   1:  PR[91,1] = PR[90,1] + 61.164;
   1:  PR[91,2] = PR[90,2] + 21.945;
   1:  PR[91,3] = PR[90,3] + 50.464;
   1:L PR[91] R[100]mm/sec CNT100;
   1:  PR[91,1] = PR[90,1] + 56.960;
   1:  PR[91,2] = PR[90,2] + 21.928;
   1:  PR[91,3] = PR[90,3] + 50.481;
   1:L PR[91] R[100]mm/sec CNT100;
   1:  PR[91,1] = PR[90,1] + 53.943;
   1:  PR[91,2] = PR[90,2] + 21.879;
   1:  PR[91,3] = PR[90,3] + 50.494;
   1:L PR[91] R[100]mm/sec CNT100;
   1:  PR[91,1] = PR[90,1] + 52.457;
   1:  PR[91,2] = PR[90,2] + 21.606;
   1:  PR[91,3] = PR[90,3] + 50.503;
   1:L PR[91] R[100]mm/sec CNT100;
   1:  PR[91,1] = PR[90,1] + 49.778;
   1:  PR[91,2] = PR[90,2] + 21.066;
   1:  PR[91,3] = PR[90,3] + 50.508;
   1:L PR[91] R[100]mm/sec CNT100;
   1:  PR[91,1] = PR[90,1] + 46.710;
   1:  PR[91,2] = PR[90,2] + 20.523;
   1:  PR[91,3] = PR[90,3] + 50.516;
   1:L PR[91] R[100]mm/sec CNT100;
   1:  PR[91,1] = PR[90,1] + 43.853;
   1:  PR[91,2] = PR[90,2] + 19.585;
   1:  PR[91,3] = PR[90,3] + 50.526;
   1:L PR[91] R[100]mm/sec CNT100;
   1:  PR[91,1] = PR[90,1] + 41.592;
   1:  PR[91,2] = PR[90,2] + 18.760;
   1:  PR[91,3] = PR[90,3] + 50.535;
   1:L PR[91] R[100]mm/sec CNT100;
   1:  PR[91,1] = PR[90,1] + 39.923;
   1:  PR[91,2] = PR[90,2] + 17.922;
   1:  PR[91,3] = PR[90,3] + 50.543;
   1:L PR[91] R[100]mm/sec CNT100;
   1:  PR[91,1] = PR[90,1] + 36.741;
   1:  PR[91,2] = PR[90,2] + 16.511;
   1:  PR[91,3] = PR[90,3] + 50.548;
   1:L PR[91] R[100]mm/sec CNT100;
   1:  PR[91,1] = PR[90,1] + 35.316;
   1:  PR[91,2] = PR[90,2] + 17.539;
   1:  PR[91,3] = PR[90,3] + 50.559;
   1:L PR[91] R[100]mm/sec CNT100;
   1:  PR[91,1] = PR[90,1] + 34.581;
   1:  PR[91,2] = PR[90,2] + 18.023;
   1:  PR[91,3] = PR[90,3] + 50.564;
   1:L PR[91] R[100]mm/sec CNT100;
   1:  PR[91,1] = PR[90,1] + 30.016;
   1:  PR[91,2] = PR[90,2] + 20.168;
   1:  PR[91,3] = PR[90,3] + 50.567;
   1:L PR[91] R[100]mm/sec CNT100;
   1:  PR[91,1] = PR[90,1] + 29.552;
   1:  PR[91,2] = PR[90,2] + 20.358;
   1:  PR[91,3] = PR[90,3] + 50.583;
   1:L PR[91] R[100]mm/sec CNT100;
   1:  PR[91,1] = PR[90,1] + 24.459;
   1:  PR[91,2] = PR[90,2] + 21.346;
   1:  PR[91,3] = PR[90,3] + 50.584;
   1:L PR[91] R[100]mm/sec CNT100;
   1:  PR[91,1] = PR[90,1] + 24.163;
   1:  PR[91,2] = PR[90,2] + 21.385;
   1:  PR[91,3] = PR[90,3] + 50.600;
   1:L PR[91] R[100]mm/sec CNT100;
   1:  PR[91,1] = PR[90,1] + 18.769;
   1:  PR[91,2] = PR[90,2] + 21.076;
   1:  PR[91,3] = PR[90,3] + 50.601;
   1:L PR[91] R[100]mm/sec CNT100;
   1:  PR[91,1] = PR[90,1] + 18.683;
   1:  PR[91,2] = PR[90,2] + 21.065;
   1:  PR[91,3] = PR[90,3] + 50.618;
   1:L PR[91] R[100]mm/sec CNT100;
   1:  PR[91,1] = PR[90,1] + 13.407;
   1:  PR[91,2] = PR[90,2] + 19.396;
   1:L PR[91] R[100]mm/sec CNT100;
   1:  PR[91,1] = PR[90,1] + 8.679;
   1:  PR[91,2] = PR[90,2] + 16.459;
   1:  PR[91,3] = PR[90,3] + 50.635;
   1:L PR[91] R[100]mm/sec CNT100;
   1:  PR[91,1] = PR[90,1] + 3.468;
   1:  PR[91,2] = PR[90,2] + 11.060;
   1:  PR[91,3] = PR[90,3] + 50.652;
   1:L PR[91] R[100]mm/sec CNT100;
   1:  PR[91,1] = PR[90,1] + -0.608;
   1:  PR[91,2] = PR[90,2] + 15.017;
   1:  PR[91,3] = PR[90,3] + 50.675;
   1:L PR[91] R[100]mm/sec CNT100;
   1:  PR[91,1] = PR[90,1] + -4.794;
   1:  PR[91,2] = PR[90,2] + 17.594;
   1:  PR[91,3] = PR[90,3] + 50.692;
   1:L PR[91] R[100]mm/sec CNT100;
   1:  PR[91,1] = PR[90,1] + -5.125;
   1:  PR[91,2] = PR[90,2] + 17.813;
   1:  PR[91,3] = PR[90,3] + 50.708;
   1:L PR[91] R[100]mm/sec CNT100;
   1:  PR[91,1] = PR[90,1] + -9.815;
   1:  PR[91,2] = PR[90,2] + 19.591;
   1:  PR[91,3] = PR[90,3] + 50.709;
   1:L PR[91] R[100]mm/sec CNT100;
   1:  PR[91,1] = PR[90,1] + -10.656;
   1:  PR[91,2] = PR[90,2] + 19.779;
   1:  PR[91,3] = PR[90,3] + 50.724;
   1:L PR[91] R[100]mm/sec CNT100;
   1:  PR[91,1] = PR[90,1] + -14.639;
   1:  PR[91,2] = PR[90,2] + 20.355;
   1:  PR[91,3] = PR[90,3] + 50.727;
   1:L PR[91] R[100]mm/sec CNT100;
   1:  PR[91,1] = PR[90,1] + -16.440;
   1:  PR[91,2] = PR[90,2] + 20.373;
   1:  PR[91,3] = PR[90,3] + 50.739;
   1:L PR[91] R[100]mm/sec CNT100;
   1:  PR[91,1] = PR[90,1] + -19.449;
   1:  PR[91,2] = PR[90,2] + 20.166;
   1:  PR[91,3] = PR[90,3] + 50.745;
   1:L PR[91] R[100]mm/sec CNT100;
   1:  PR[91,1] = PR[90,1] + -22.024;
   1:  PR[91,2] = PR[90,2] + 19.650;
   1:  PR[91,3] = PR[90,3] + 50.754;
   1:L PR[91] R[100]mm/sec CNT100;
   1:  PR[91,1] = PR[90,1] + -24.055;
   1:  PR[91,2] = PR[90,2] + 19.067;
   1:  PR[91,3] = PR[90,3] + 50.762;
   1:L PR[91] R[100]mm/sec CNT100;
   1:  PR[91,1] = PR[90,1] + -27.088;
   1:  PR[91,2] = PR[90,2] + 17.767;
   1:  PR[91,3] = PR[90,3] + 50.769;
   1:L PR[91] R[100]mm/sec CNT100;
   1:  PR[91,1] = PR[90,1] + -28.281;
   1:  PR[91,2] = PR[90,2] + 17.128;
   1:  PR[91,3] = PR[90,3] + 50.779;
   1:L PR[91] R[100]mm/sec CNT100;
   1:  PR[91,1] = PR[90,1] + -31.804;
   1:  PR[91,2] = PR[90,2] + 14.640;
   1:  PR[91,3] = PR[90,3] + 50.783;
   1:L PR[91] R[100]mm/sec CNT100;
   1:  PR[91,1] = PR[90,1] + -32.077;
   1:  PR[91,2] = PR[90,2] + 14.400;
   1:  PR[91,3] = PR[90,3] + 50.796;
   1:L PR[91] R[100]mm/sec CNT100;
   1:  PR[91,1] = PR[90,1] + -32.371;
   1:  PR[91,2] = PR[90,2] + 14.116;
   1:  PR[91,3] = PR[90,3] + 50.797;
   1:L PR[91] R[100]mm/sec CNT100;
   1:  PR[91,1] = PR[90,1] + -35.672;
   1:  PR[91,2] = PR[90,2] + 10.579;
   1:  PR[91,3] = PR[90,3] + 50.798;
   1:L PR[91] R[100]mm/sec CNT100;
   1:  PR[91,1] = PR[90,1] + -39.359;
   1:  PR[91,2] = PR[90,2] + 13.056;
   1:  PR[91,3] = PR[90,3] + 50.813;
   1:L PR[91] R[100]mm/sec CNT100;
   1:  PR[91,1] = PR[90,1] + -40.947;
   1:  PR[91,2] = PR[90,2] + 14.339;
   1:  PR[91,3] = PR[90,3] + 50.827;
   1:L PR[91] R[100]mm/sec CNT100;
   1:  PR[91,1] = PR[90,1] + -41.655;
   1:  PR[91,2] = PR[90,2] + 14.865;
   1:  PR[91,3] = PR[90,3] + 50.833;
   1:L PR[91] R[100]mm/sec CNT100;
   1:  PR[91,1] = PR[90,1] + -44.491;
   1:  PR[91,2] = PR[90,2] + 16.278;
   1:  PR[91,3] = PR[90,3] + 50.836;
   1:L PR[91] R[100]mm/sec CNT100;
   1:  PR[91,1] = PR[90,1] + -47.745;
   1:  PR[91,2] = PR[90,2] + 17.786;
   1:  PR[91,3] = PR[90,3] + 50.846;
   1:L PR[91] R[100]mm/sec CNT100;
   1:  PR[91,1] = PR[90,1] + -49.480;
   1:  PR[91,2] = PR[90,2] + 18.254;
   1:  PR[91,3] = PR[90,3] + 50.857;
   1:L PR[91] R[100]mm/sec CNT100;
   1:  PR[91,1] = PR[90,1] + -52.593;
   1:  PR[91,2] = PR[90,2] + 19.203;
   1:  PR[91,3] = PR[90,3] + 50.862;
   1:L PR[91] R[100]mm/sec CNT100;
   1:  PR[91,1] = PR[90,1] + -53.909;
   1:  PR[91,2] = PR[90,2] + 19.567;
   1:  PR[91,3] = PR[90,3] + 50.872;
   1:L PR[91] R[100]mm/sec CNT100;
   1:  PR[91,1] = PR[90,1] + -56.609;
   1:  PR[91,2] = PR[90,2] + 19.882;
   1:  PR[91,3] = PR[90,3] + 50.876;
   1:L PR[91] R[100]mm/sec CNT100;
   1:  PR[91,1] = PR[90,1] + -59.914;
   1:  PR[91,2] = PR[90,2] + 20.201;
   1:  PR[91,3] = PR[90,3] + 50.885;
   1:L PR[91] R[100]mm/sec CNT100;
   1:  PR[91] = PR[90];
   1:  PR[91,1] = PR[90,1] + -64.669;
   1:  PR[91,2] = PR[90,2] + 19.991;
   1:  PR[91,3] = PR[90,3] + 52.195;
   1:L PR[91] R[100]mm/sec CNT100;
   1:  PR[91,1] = PR[90,1] + -69.564;
   1:  PR[91,2] = PR[90,2] + 18.776;
   1:  PR[91,3] = PR[90,3] + 50.908;
   1:L PR[91] R[100]mm/sec CNT100;
   1:  PR[91,1] = PR[90,1] + -73.967;
   1:  PR[91,2] = PR[90,2] + 16.786;
   1:  PR[91,3] = PR[90,3] + 50.924;
   1:L PR[91] R[100]mm/sec CNT100;
   1:  PR[91,1] = PR[90,1] + -76.287;
   1:  PR[91,2] = PR[90,2] + 15.170;
   1:  PR[91,3] = PR[90,3] + 50.939;
   1:L PR[91] R[100]mm/sec CNT100;
   1:  PR[91,1] = PR[90,1] + -77.765;
   1:  PR[91,2] = PR[90,2] + 14.124;
   1:  PR[91,3] = PR[90,3] + 50.947;
   1:L PR[91] R[100]mm/sec CNT100;
   1:  PR[91,1] = PR[90,1] + -80.847;
   1:  PR[91,2] = PR[90,2] + 10.897;
   1:  PR[91,3] = PR[90,3] + 50.953;
   1:L PR[91] R[100]mm/sec CNT100;
   1:  PR[91,1] = PR[90,1] + -83.109;
   1:  PR[91,2] = PR[90,2] + 7.254;
   1:  PR[91,3] = PR[90,3] + 50.967;
   1:L PR[91] R[100]mm/sec CNT100;
   1:  PR[91,1] = PR[90,1] + -84.487;
   1:  PR[91,2] = PR[90,2] + 3.334;
   1:  PR[91,3] = PR[90,3] + 50.980;
   1:L PR[91] R[100]mm/sec CNT100;
   1:  PR[91,1] = PR[90,1] + -84.931;
   1:  PR[91,2] = PR[90,2] + -0.663;
   1:  PR[91,3] = PR[90,3] + 50.993;
   1:L PR[91] R[100]mm/sec CNT100;
   1:  PR[91,1] = PR[90,1] + -84.602;
   1:  PR[91,2] = PR[90,2] + -2.181;
   1:  PR[91,3] = PR[90,3] + 51.006;
   1:L PR[91] R[100]mm/sec CNT100;
   1:  PR[91,1] = PR[90,1] + -84.313;
   1:  PR[91,2] = PR[90,2] + -4.806;
   1:  PR[91,3] = PR[90,3] + 51.010;
   1:L PR[91] R[100]mm/sec CNT100;
   1:  PR[91,1] = PR[90,1] + -83.840;
   1:  PR[91,2] = PR[90,2] + -6.180;
   1:  PR[91,3] = PR[90,3] + 51.019;
   1:L PR[91] R[100]mm/sec CNT100;
   1:  PR[91,1] = PR[90,1] + -82.971;
   1:  PR[91,2] = PR[90,2] + -8.742;
   1:  PR[91,3] = PR[90,3] + 51.023;
   1:L PR[91] R[100]mm/sec CNT100;
   1:  PR[91,1] = PR[90,1] + -80.777;
   1:  PR[91,2] = PR[90,2] + -12.383;
   1:  PR[91,3] = PR[90,3] + 51.032;
   1:L PR[91] R[100]mm/sec CNT100;
   1:  PR[91,1] = PR[90,1] + -77.798;
   1:  PR[91,2] = PR[90,2] + -15.593;
   1:  PR[91,3] = PR[90,3] + 51.045;
   1:L PR[91] R[100]mm/sec CNT100;
   1:  PR[91,1] = PR[90,1] + -74.972;
   1:  PR[91,2] = PR[90,2] + -17.625;
   1:  PR[91,3] = PR[90,3] + 51.058;
   1:L PR[91] R[100]mm/sec CNT100;
   1:  PR[91,1] = PR[90,1] + -74.110;
   1:  PR[91,2] = PR[90,2] + -18.218;
   1:  PR[91,3] = PR[90,3] + 51.069;
   1:L PR[91] R[100]mm/sec CNT100;
   1:  PR[91,1] = PR[90,1] + -74.072;
   1:  PR[91,2] = PR[90,2] + -18.242;
   1:  PR[91,3] = PR[90,3] + 51.072;
   1:L PR[91] R[100]mm/sec CNT100;
   1:  PR[91,1] = PR[90,1] + -70.237;
   1:  PR[91,2] = PR[90,2] + -19.943;
   1:  PR[91,3] = PR[90,3] + 51.073;
   1:L PR[91] R[100]mm/sec CNT100;
   1:  PR[91,1] = PR[90,1] + -69.060;
   1:  PR[91,2] = PR[90,2] + -20.391;
   1:  PR[91,3] = PR[90,3] + 51.086;
   1:L PR[91] R[100]mm/sec CNT100;
   1:  PR[91,1] = PR[90,1] + -66.020;
   1:  PR[91,2] = PR[90,2] + -21.135;
   1:  PR[91,3] = PR[90,3] + 51.090;
   1:L PR[91] R[100]mm/sec CNT100;
   1:  PR[91,1] = PR[90,1] + -63.204;
   1:  PR[91,2] = PR[90,2] + -21.637;
   1:  PR[91,3] = PR[90,3] + 51.099;
   1:L PR[91] R[100]mm/sec CNT100;
   1:  PR[91,1] = PR[90,1] + -61.535;
   1:  PR[91,2] = PR[90,2] + -21.748;
   1:  PR[91,3] = PR[90,3] + 51.108;
   1:L PR[91] R[100]mm/sec CNT100;
   1:  PR[91,1] = PR[90,1] + -56.702;
   1:  PR[91,2] = PR[90,2] + -21.708;
   1:  PR[91,3] = PR[90,3] + 51.113;
   1:L PR[91] R[100]mm/sec CNT100;
   1:  PR[91,1] = PR[90,1] + -50.491;
   1:  PR[91,2] = PR[90,2] + -20.719;
   1:  PR[91,3] = PR[90,3] + 51.128;
   1:L PR[91] R[100]mm/sec CNT100;
   1:  PR[91,1] = PR[90,1] + -44.607;
   1:  PR[91,2] = PR[90,2] + -18.703;
   1:  PR[91,3] = PR[90,3] + 51.148;
   1:L PR[91] R[100]mm/sec CNT100;
   1:  PR[91,1] = PR[90,1] + -43.795;
   1:  PR[91,2] = PR[90,2] + -18.231;
   1:  PR[91,3] = PR[90,3] + 51.167;
   1:L PR[91] R[100]mm/sec CNT100;
   1:  PR[91,1] = PR[90,1] + -39.900;
   1:  PR[91,2] = PR[90,2] + -16.332;
   1:  PR[91,3] = PR[90,3] + 51.170;
   1:L PR[91] R[100]mm/sec CNT100;
   1:  PR[91,1] = PR[90,1] + -37.643;
   1:  PR[91,2] = PR[90,2] + -15.012;
   1:  PR[91,3] = PR[90,3] + 51.184;
   1:L PR[91] R[100]mm/sec CNT100;
   1:  PR[91,1] = PR[90,1] + -34.795;
   1:  PR[91,2] = PR[90,2] + -12.750;
   1:  PR[91,3] = PR[90,3] + 51.192;
   1:L PR[91] R[100]mm/sec CNT100;
   1:  PR[91,1] = PR[90,1] + -32.375;
   1:  PR[91,2] = PR[90,2] + -15.360;
   1:  PR[91,3] = PR[90,3] + 51.203;
   1:L PR[91] R[100]mm/sec CNT100;
   1:  PR[91,1] = PR[90,1] + -32.046;
   1:  PR[91,2] = PR[90,2] + -15.679;
   1:  PR[91,3] = PR[90,3] + 51.214;
   1:L PR[91] R[100]mm/sec CNT100;
   1:  PR[91,1] = PR[90,1] + -30.967;
   1:  PR[91,2] = PR[90,2] + -16.576;
   1:  PR[91,3] = PR[90,3] + 51.215;
   1:L PR[91] R[100]mm/sec CNT100;
   1:  PR[91,1] = PR[90,1] + -28.364;
   1:  PR[91,2] = PR[90,2] + -18.417;
   1:  PR[91,3] = PR[90,3] + 51.220;
   1:L PR[91] R[100]mm/sec CNT100;
   1:  PR[91,1] = PR[90,1] + -28.142;
   1:  PR[91,2] = PR[90,2] + -18.564;
   1:  PR[91,3] = PR[90,3] + 51.230;
   1:L PR[91] R[100]mm/sec CNT100;
   1:  PR[91,1] = PR[90,1] + -26.377;
   1:  PR[91,2] = PR[90,2] + -19.515;
   1:  PR[91,3] = PR[90,3] + 51.231;
   1:L PR[91] R[100]mm/sec CNT100;
   1:  PR[91,1] = PR[90,1] + -23.862;
   1:  PR[91,2] = PR[90,2] + -20.594;
   1:  PR[91,3] = PR[90,3] + 51.237;
   1:L PR[91] R[100]mm/sec CNT100;
   1:  PR[91,1] = PR[90,1] + -21.221;
   1:  PR[91,2] = PR[90,2] + -21.357;
   1:  PR[91,3] = PR[90,3] + 51.245;
   1:L PR[91] R[100]mm/sec CNT100;
   1:  PR[91,1] = PR[90,1] + -19.235;
   1:  PR[91,2] = PR[90,2] + -21.756;
   1:  PR[91,3] = PR[90,3] + 51.254;
   1:L PR[91] R[100]mm/sec CNT100;
   1:  PR[91,1] = PR[90,1] + -15.550;
   1:  PR[91,2] = PR[90,2] + -22.015;
   1:  PR[91,3] = PR[90,3] + 51.260;
   1:L PR[91] R[100]mm/sec CNT100;
   1:  PR[91,1] = PR[90,1] + -14.387;
   1:  PR[91,2] = PR[90,2] + -22.004;
   1:  PR[91,3] = PR[90,3] + 51.272;
   1:L PR[91] R[100]mm/sec CNT100;
   1:  PR[91,1] = PR[90,1] + -9.688;
   1:  PR[91,2] = PR[90,2] + -21.331;
   1:  PR[91,3] = PR[90,3] + 51.275;
   1:L PR[91] R[100]mm/sec CNT100;
   1:  PR[91,1] = PR[90,1] + -9.508;
   1:  PR[91,2] = PR[90,2] + -21.291;
   1:  PR[91,3] = PR[90,3] + 51.290;
   1:L PR[91] R[100]mm/sec CNT100;
   1:  PR[91,1] = PR[90,1] + -7.554;
   1:  PR[91,2] = PR[90,2] + -20.556;
   1:L PR[91] R[100]mm/sec CNT100;
   1:  PR[91,1] = PR[90,1] + -4.420;
   1:  PR[91,2] = PR[90,2] + -19.477;
   1:  PR[91,3] = PR[90,3] + 51.297;
   1:L PR[91] R[100]mm/sec CNT100;
   1:  PR[91,1] = PR[90,1] + -3.858;
   1:  PR[91,2] = PR[90,2] + -19.154;
   1:  PR[91,3] = PR[90,3] + 51.307;
   1:L PR[91] R[100]mm/sec CNT100;
   1:  PR[91,1] = PR[90,1] + 0.098;
   1:  PR[91,2] = PR[90,2] + -16.727;
   1:  PR[91,3] = PR[90,3] + 51.309;
   1:L PR[91] R[100]mm/sec CNT100;
   1:  PR[91,1] = PR[90,1] + 1.532;
   1:  PR[91,2] = PR[90,2] + -15.397;
   1:  PR[91,3] = PR[90,3] + 51.324;
   1:L PR[91] R[100]mm/sec CNT100;
   1:  PR[91,1] = PR[90,1] + 6.706;
   1:  PR[91,2] = PR[90,2] + -10.230;
   1:  PR[91,3] = PR[90,3] + 51.330;
   1:L PR[91] R[100]mm/sec CNT100;
   1:  PR[91,1] = PR[90,1] + 5.778;
   1:  PR[91,2] = PR[90,2] + -15.484;
   1:  PR[91,3] = PR[90,3] + 51.352;
   1:L PR[91] R[100]mm/sec CNT100;
   1:  PR[91,1] = PR[90,1] + 6.415;
   1:  PR[91,2] = PR[90,2] + -16.143;
   1:  PR[91,3] = PR[90,3] + 51.369;
   1:L PR[91] R[100]mm/sec CNT100;
   1:  PR[91,1] = PR[90,1] + 8.261;
   1:  PR[91,2] = PR[90,2] + -17.974;
   1:  PR[91,3] = PR[90,3] + 51.372;
   1:L PR[91] R[100]mm/sec CNT100;
   1:  PR[91,1] = PR[90,1] + 8.430;
   1:  PR[91,2] = PR[90,2] + -18.113;
   1:  PR[91,3] = PR[90,3] + 51.380;
   1:L PR[91] R[100]mm/sec CNT100;
   1:  PR[91,1] = PR[90,1] + 13.025;
   1:  PR[91,2] = PR[90,2] + -20.955;
   1:  PR[91,3] = PR[90,3] + 51.381;
   1:L PR[91] R[100]mm/sec CNT100;
   1:  PR[91,1] = PR[90,1] + 13.198;
   1:  PR[91,2] = PR[90,2] + -21.049;
   1:  PR[91,3] = PR[90,3] + 51.397;
   1:L PR[91] R[100]mm/sec CNT100;
   1:  PR[91,1] = PR[90,1] + 18.562;
   1:  PR[91,2] = PR[90,2] + -22.720;
   1:  PR[91,3] = PR[90,3] + 51.398;
   1:L PR[91] R[100]mm/sec CNT100;
   1:  PR[91,1] = PR[90,1] + 24.134;
   1:  PR[91,2] = PR[90,2] + -23.029;
   1:  PR[91,3] = PR[90,3] + 51.416;
   1:L PR[91] R[100]mm/sec CNT100;
   1:  PR[91,1] = PR[90,1] + 29.605;
   1:  PR[91,2] = PR[90,2] + -21.970;
   1:  PR[91,3] = PR[90,3] + 51.433;
   1:L PR[91] R[100]mm/sec CNT100;
   1:  PR[91,1] = PR[90,1] + 34.594;
   1:  PR[91,2] = PR[90,2] + -19.626;
   1:  PR[91,3] = PR[90,3] + 51.450;
   1:L PR[91] R[100]mm/sec CNT100;
   1:  PR[91,1] = PR[90,1] + 34.874;
   1:  PR[91,2] = PR[90,2] + -19.413;
   1:  PR[91,3] = PR[90,3] + 51.467;
   1:L PR[91] R[100]mm/sec CNT100;
   1:  PR[91,1] = PR[90,1] + 36.178;
   1:  PR[91,2] = PR[90,2] + -18.696;
   1:  PR[91,3] = PR[90,3] + 51.468;
   1:L PR[91] R[100]mm/sec CNT100;
   1:  PR[91,1] = PR[90,1] + 40.181;
   1:  PR[91,2] = PR[90,2] + -20.483;
   1:  PR[91,3] = PR[90,3] + 51.473;
   1:L PR[91] R[100]mm/sec CNT100;
   1:  PR[91,1] = PR[90,1] + 40.675;
   1:  PR[91,2] = PR[90,2] + -20.685;
   1:  PR[91,3] = PR[90,3] + 51.487;
   1:L PR[91] R[100]mm/sec CNT100;
   1:  PR[91,1] = PR[90,1] + 45.542;
   1:  PR[91,2] = PR[90,2] + -22.276;
   1:  PR[91,3] = PR[90,3] + 51.488;
   1:L PR[91] R[100]mm/sec CNT100;
   1:  PR[91,1] = PR[90,1] + 51.283;
   1:  PR[91,2] = PR[90,2] + -23.296;
   1:  PR[91,3] = PR[90,3] + 51.504;
   1:L PR[91] R[100]mm/sec CNT100;
   1:  PR[91,1] = PR[90,1] + 52.686;
   1:  PR[91,2] = PR[90,2] + -23.569;
   1:  PR[91,3] = PR[90,3] + 51.522;
   1:L PR[91] R[100]mm/sec CNT100;
   1:  PR[91,1] = PR[90,1] + 56.817;
   1:  PR[91,2] = PR[90,2] + -23.644;
   1:  PR[91,3] = PR[90,3] + 51.527;
   1:L PR[91] R[100]mm/sec CNT100;
   1:  PR[91,1] = PR[90,1] + 60.086;
   1:  PR[91,2] = PR[90,2] + -23.648;
   1:  PR[91,3] = PR[90,3] + 51.540;
   1:L PR[91] R[100]mm/sec CNT100;
   1:  PR[91,1] = PR[90,1] + 61.434;
   1:  PR[91,2] = PR[90,2] + -23.431;
   1:  PR[91,3] = PR[90,3] + 51.550;
   1:L PR[91] R[100]mm/sec CNT100;
   1:  PR[91,1] = PR[90,1] + 66.415;
   1:  PR[91,2] = PR[90,2] + -22.564;
   1:  PR[91,3] = PR[90,3] + 51.554;
   1:L PR[91] R[100]mm/sec CNT100;
   1:  PR[91,1] = PR[90,1] + 67.092;
   1:  PR[91,2] = PR[90,2] + -22.360;
   1:  PR[91,3] = PR[90,3] + 51.570;
   1:L PR[91] R[100]mm/sec CNT100;
   1:  PR[91,1] = PR[90,1] + 71.318;
   1:  PR[91,2] = PR[90,2] + -20.761;
   1:  PR[91,3] = PR[90,3] + 51.572;
   1:L PR[91] R[100]mm/sec CNT100;
   1:  PR[91,1] = PR[90,1] + 73.844;
   1:  PR[91,2] = PR[90,2] + -19.387;
   1:  PR[91,3] = PR[90,3] + 51.586;
   1:L PR[91] R[100]mm/sec CNT100;
   1:  PR[91,1] = PR[90,1] + 75.892;
   1:  PR[91,2] = PR[90,2] + -18.107;
   1:  PR[91,3] = PR[90,3] + 51.595;
   1:L PR[91] R[100]mm/sec CNT100;
   1:  PR[91,1] = PR[90,1] + 79.223;
   1:  PR[91,2] = PR[90,2] + -15.223;
   1:  PR[91,3] = PR[90,3] + 51.602;
   1:L PR[91] R[100]mm/sec CNT100;
   1:  PR[91,1] = PR[90,1] + 79.845;
   1:  PR[91,2] = PR[90,2] + -14.627;
   1:  PR[91,3] = PR[90,3] + 51.616;
   1:L PR[91] R[100]mm/sec CNT100;
   1:  PR[91,1] = PR[90,1] + 82.912;
   1:  PR[91,2] = PR[90,2] + -10.395;
   1:  PR[91,3] = PR[90,3] + 51.619;
   1:L PR[91] R[100]mm/sec CNT100;
   1:  PR[91,1] = PR[90,1] + 83.185;
   1:  PR[91,2] = PR[90,2] + -9.720;
   1:  PR[91,3] = PR[90,3] + 51.635;
   1:L PR[91] R[100]mm/sec CNT100;
   1:  PR[91,1] = PR[90,1] + 84.744;
   1:  PR[91,2] = PR[90,2] + -5.669;
   1:  PR[91,3] = PR[90,3] + 51.637;
   1:L PR[91] R[100]mm/sec CNT100;
   1:  PR[91,1] = PR[90,1] + 85.358;
   1:  PR[91,2] = PR[90,2] + -0.729;
   1:  PR[91,3] = PR[90,3] + 51.651;
   1:L PR[91] R[100]mm/sec CNT100;
   1:  PR[91,1] = PR[90,1] + 84.744;
   1:  PR[91,2] = PR[90,2] + 4.210;
   1:  PR[91,3] = PR[90,3] + 51.666;
   1:L PR[91] R[100]mm/sec CNT100;
   1:  PR[91,1] = PR[90,1] + 83.185;
   1:  PR[91,2] = PR[90,2] + 8.261;
   1:  PR[91,3] = PR[90,3] + 51.682;
   1:L PR[91] R[100]mm/sec CNT100;
   1:  PR[91,1] = PR[90,1] + 82.912;
   1:  PR[91,2] = PR[90,2] + 8.936;
   1:  PR[91,3] = PR[90,3] + 51.695;
   1:L PR[91] R[100]mm/sec CNT100;
   1:  PR[91,1] = PR[90,1] + 79.843;
   1:  PR[91,2] = PR[90,2] + 13.170;
   1:  PR[91,3] = PR[90,3] + 51.697;
   1:L PR[91] R[100]mm/sec CNT100;
   1:  PR[91,1] = PR[90,1] + 79.217;
   1:  PR[91,2] = PR[90,2] + 13.769;
   1:  PR[91,3] = PR[90,3] + 51.714;
   1:L PR[91] R[100]mm/sec CNT100;
   1:  PR[91,1] = PR[90,1] + 75.883;
   1:  PR[91,2] = PR[90,2] + 16.655;
   1:  PR[91,3] = PR[90,3] + 51.716;
   1:L PR[91] R[100]mm/sec CNT100;
   1:  PR[91,1] = PR[90,1] + 73.820;
   1:  PR[91,2] = PR[90,2] + 17.941;
   1:  PR[91,3] = PR[90,3] + 51.730;
   1:L PR[91] R[100]mm/sec CNT100;
   1:  PR[91,1] = PR[90,1] + 71.296;
   1:  PR[91,2] = PR[90,2] + 19.314;
   1:  PR[91,3] = PR[90,3] + 51.737;
   1:L PR[91] R[100]mm/sec CNT100;
   1:  PR[91,1] = PR[90,1] + 67.030;
   1:  PR[91,2] = PR[90,2] + 20.920;
   1:  PR[91,3] = PR[90,3] + 51.746;
   1:L PR[91] R[100]mm/sec CNT100;
   1:  PR[91,1] = PR[90,1] + 66.371;
   1:  PR[91,2] = PR[90,2] + 21.117;
   1:  PR[91,3] = PR[90,3] + 51.761;
   1:L PR[91] R[100]mm/sec CNT100;
   1:  PR[91,1] = PR[90,1] + 61.393;
   1:  PR[91,2] = PR[90,2] + 21.973;
   1:  PR[91,3] = PR[90,3] + 51.763;
   1:L PR[91] R[100]mm/sec CNT100;
   1:  PR[91,1] = PR[90,1] + 60.040;
   1:  PR[91,2] = PR[90,2] + 22.193;
   1:  PR[91,3] = PR[90,3] + 51.778;
   1:L PR[91] R[100]mm/sec CNT100;
   1:  PR[91,1] = PR[90,1] + 56.801;
   1:  PR[91,2] = PR[90,2] + 22.180;
   1:  PR[91,3] = PR[90,3] + 51.783;
   1:L PR[91] R[100]mm/sec CNT100;
   1:  PR[91,1] = PR[90,1] + 52.708;
   1:  PR[91,2] = PR[90,2] + 22.112;
   1:  PR[91,3] = PR[90,3] + 51.793;
   1:L PR[91] R[100]mm/sec CNT100;
   1:  PR[91,1] = PR[90,1] + 51.286;
   1:  PR[91,2] = PR[90,2] + 21.836;
   1:  PR[91,3] = PR[90,3] + 51.805;
   1:L PR[91] R[100]mm/sec CNT100;
   1:  PR[91,1] = PR[90,1] + 47.274;
   1:  PR[91,2] = PR[90,2] + 21.109;
   1:  PR[91,3] = PR[90,3] + 51.810;
   1:L PR[91] R[100]mm/sec CNT100;
   1:  PR[91,1] = PR[90,1] + 45.552;
   1:  PR[91,2] = PR[90,2] + 20.819;
   1:  PR[91,3] = PR[90,3] + 51.823;
   1:L PR[91] R[100]mm/sec CNT100;
   1:  PR[91,1] = PR[90,1] + 40.675;
   1:  PR[91,2] = PR[90,2] + 19.227;
   1:  PR[91,3] = PR[90,3] + 51.828;
   1:L PR[91] R[100]mm/sec CNT100;
   1:  PR[91,1] = PR[90,1] + 40.181;
   1:  PR[91,2] = PR[90,2] + 19.024;
   1:  PR[91,3] = PR[90,3] + 51.844;
   1:L PR[91] R[100]mm/sec CNT100;
   1:  PR[91,1] = PR[90,1] + 36.085;
   1:  PR[91,2] = PR[90,2] + 17.196;
   1:  PR[91,3] = PR[90,3] + 51.846;
   1:L PR[91] R[100]mm/sec CNT100;
   1:  PR[91,1] = PR[90,1] + 34.652;
   1:  PR[91,2] = PR[90,2] + 18.140;
   1:  PR[91,3] = PR[90,3] + 51.860;
   1:L PR[91] R[100]mm/sec CNT100;
   1:  PR[91,1] = PR[90,1] + 29.608;
   1:  PR[91,2] = PR[90,2] + 20.510;
   1:  PR[91,3] = PR[90,3] + 51.865;
   1:L PR[91] R[100]mm/sec CNT100;
   1:  PR[91,1] = PR[90,1] + 24.139;
   1:  PR[91,2] = PR[90,2] + 21.570;
   1:  PR[91,3] = PR[90,3] + 51.882;
   1:L PR[91] R[100]mm/sec CNT100;
   1:  PR[91,1] = PR[90,1] + 18.570;
   1:  PR[91,2] = PR[90,2] + 21.262;
   1:  PR[91,3] = PR[90,3] + 51.899;
   1:L PR[91] R[100]mm/sec CNT100;
   1:  PR[91,1] = PR[90,1] + 13.208;
   1:  PR[91,2] = PR[90,2] + 19.594;
   1:  PR[91,3] = PR[90,3] + 51.917;
   1:L PR[91] R[100]mm/sec CNT100;
   1:  PR[91,1] = PR[90,1] + 13.032;
   1:  PR[91,2] = PR[90,2] + 19.499;
   1:  PR[91,3] = PR[90,3] + 51.934;
   1:L PR[91] R[100]mm/sec CNT100;
   1:  PR[91,1] = PR[90,1] + 8.439;
   1:  PR[91,2] = PR[90,2] + 16.662;
   1:  PR[91,3] = PR[90,3] + 51.935;
   1:L PR[91] R[100]mm/sec CNT100;
   1:  PR[91,1] = PR[90,1] + 8.239;
   1:  PR[91,2] = PR[90,2] + 16.497;
   1:  PR[91,3] = PR[90,3] + 51.952;
   1:L PR[91] R[100]mm/sec CNT100;
   1:  PR[91,1] = PR[90,1] + 8.062;
   1:  PR[91,2] = PR[90,2] + 16.331;
   1:L PR[91] R[100]mm/sec CNT100;
   1:  PR[91,1] = PR[90,1] + 3.688;
   1:  PR[91,2] = PR[90,2] + 11.788;
   1:  PR[91,3] = PR[90,3] + 51.953;
   1:L PR[91] R[100]mm/sec CNT100;
   1:  PR[91,1] = PR[90,1] + 0.251;
   1:  PR[91,2] = PR[90,2] + 15.141;
   1:  PR[91,3] = PR[90,3] + 51.973;
   1:L PR[91] R[100]mm/sec CNT100;
   1:  PR[91,1] = PR[90,1] + 0.146;
   1:  PR[91,2] = PR[90,2] + 15.233;
   1:  PR[91,3] = PR[90,3] + 51.988;
   1:L PR[91] R[100]mm/sec CNT100;
   1:  PR[91,1] = PR[90,1] + -3.815;
   1:  PR[91,2] = PR[90,2] + 17.671;
   1:L PR[91] R[100]mm/sec CNT100;
   1:  PR[91,1] = PR[90,1] + -4.394;
   1:  PR[91,2] = PR[90,2] + 18.005;
   1:  PR[91,3] = PR[90,3] + 52.003;
   1:L PR[91] R[100]mm/sec CNT100;
   1:  PR[91,1] = PR[90,1] + -7.556;
   1:  PR[91,2] = PR[90,2] + 19.099;
   1:  PR[91,3] = PR[90,3] + 52.005;
   1:L PR[91] R[100]mm/sec CNT100;
   1:  PR[91,1] = PR[90,1] + -9.478;
   1:  PR[91,2] = PR[90,2] + 19.825;
   1:  PR[91,3] = PR[90,3] + 52.015;
   1:L PR[91] R[100]mm/sec CNT100;
   1:  PR[91,1] = PR[90,1] + -9.653;
   1:  PR[91,2] = PR[90,2] + 19.864;
   1:  PR[91,3] = PR[90,3] + 52.021;
   1:L PR[91] R[100]mm/sec CNT100;
   1:  PR[91,1] = PR[90,1] + -14.358;
   1:  PR[91,2] = PR[90,2] + 20.544;
   1:  PR[91,3] = PR[90,3] + 52.022;
   1:L PR[91] R[100]mm/sec CNT100;
   1:  PR[91,1] = PR[90,1] + -15.516;
   1:  PR[91,2] = PR[90,2] + 20.556;
   1:  PR[91,3] = PR[90,3] + 52.037;
   1:L PR[91] R[100]mm/sec CNT100;
   1:  PR[91,1] = PR[90,1] + -19.208;
   1:  PR[91,2] = PR[90,2] + 20.301;
   1:  PR[91,3] = PR[90,3] + 52.040;
   1:L PR[91] R[100]mm/sec CNT100;
   1:  PR[91,1] = PR[90,1] + -21.192;
   1:  PR[91,2] = PR[90,2] + 19.904;
   1:  PR[91,3] = PR[90,3] + 52.052;
   1:L PR[91] R[100]mm/sec CNT100;
   1:  PR[91,1] = PR[90,1] + -23.839;
   1:  PR[91,2] = PR[90,2] + 19.144;
   1:  PR[91,3] = PR[90,3] + 52.058;
   1:L PR[91] R[100]mm/sec CNT100;
   1:  PR[91,1] = PR[90,1] + -26.354;
   1:  PR[91,2] = PR[90,2] + 18.066;
   1:  PR[91,3] = PR[90,3] + 52.067;
   1:L PR[91] R[100]mm/sec CNT100;
   1:  PR[91,1] = PR[90,1] + -28.076;
   1:  PR[91,2] = PR[90,2] + 17.144;
   1:  PR[91,3] = PR[90,3] + 52.075;
   1:L PR[91] R[100]mm/sec CNT100;
   1:  PR[91,1] = PR[90,1] + -31.408;
   1:  PR[91,2] = PR[90,2] + 14.789;
   1:  PR[91,3] = PR[90,3] + 52.081;
   1:L PR[91] R[100]mm/sec CNT100;
   1:  PR[91,1] = PR[90,1] + -31.909;
   1:  PR[91,2] = PR[90,2] + 14.349;
   1:  PR[91,3] = PR[90,3] + 52.094;
   1:L PR[91] R[100]mm/sec CNT100;
   1:  PR[91,1] = PR[90,1] + -32.417;
   1:  PR[91,2] = PR[90,2] + 13.858;
   1:  PR[91,3] = PR[90,3] + 52.096;
   1:L PR[91] R[100]mm/sec CNT100;
   1:  PR[91,1] = PR[90,1] + -34.710;
   1:  PR[91,2] = PR[90,2] + 11.401;
   1:  PR[91,3] = PR[90,3] + 52.098;
   1:L PR[91] R[100]mm/sec CNT100;
   1:  PR[91,1] = PR[90,1] + -39.781;
   1:  PR[91,2] = PR[90,2] + 14.820;
   1:  PR[91,3] = PR[90,3] + 52.109;
   1:L PR[91] R[100]mm/sec CNT100;
   1:  PR[91,1] = PR[90,1] + -39.941;
   1:  PR[91,2] = PR[90,2] + 14.904;
   1:  PR[91,3] = PR[90,3] + 52.128;
   1:L PR[91] R[100]mm/sec CNT100;
   1:  PR[91,1] = PR[90,1] + -40.276;
   1:  PR[91,2] = PR[90,2] + 15.043;
   1:L PR[91] R[100]mm/sec CNT100;
   1:  PR[91,1] = PR[90,1] + -44.030;
   1:  PR[91,2] = PR[90,2] + 16.915;
   1:  PR[91,3] = PR[90,3] + 52.129;
   1:L PR[91] R[100]mm/sec CNT100;
   1:  PR[91,1] = PR[90,1] + -46.182;
   1:  PR[91,2] = PR[90,2] + 17.912;
   1:  PR[91,3] = PR[90,3] + 52.142;
   1:L PR[91] R[100]mm/sec CNT100;
   1:  PR[91,1] = PR[90,1] + -47.907;
   1:  PR[91,2] = PR[90,2] + 18.403;
   1:  PR[91,3] = PR[90,3] + 52.150;
   1:L PR[91] R[100]mm/sec CNT100;
   1:  PR[91,1] = PR[90,1] + -51.128;
   1:  PR[91,2] = PR[90,2] + 19.245;
   1:  PR[91,3] = PR[90,3] + 52.155;
   1:L PR[91] R[100]mm/sec CNT100;
   1:  PR[91,1] = PR[90,1] + -52.323;
   1:  PR[91,2] = PR[90,2] + 19.609;
   1:  PR[91,3] = PR[90,3] + 52.166;
   1:L PR[91] R[100]mm/sec CNT100;
   1:  PR[91,1] = PR[90,1] + -52.717;
   1:  PR[91,2] = PR[90,2] + 19.718;
   1:  PR[91,3] = PR[90,3] + 52.169;
   1:L PR[91] R[100]mm/sec CNT100;
   1:  PR[91,1] = PR[90,1] + -56.382;
   1:  PR[91,2] = PR[90,2] + 20.146;
   1:  PR[91,3] = PR[90,3] + 52.171;
   1:L PR[91] R[100]mm/sec CNT100;
   1:  PR[91,1] = PR[90,1] + -58.819;
   1:  PR[91,2] = PR[90,2] + 20.382;
   1:  PR[91,3] = PR[90,3] + 52.182;
   1:L PR[91] R[100]mm/sec CNT100;
   1:  PR[91,1] = PR[90,1] + -60.497;
   1:  PR[91,2] = PR[90,2] + 20.289;
   1:  PR[91,3] = PR[90,3] + 52.190;
   1:L PR[91] R[100]mm/sec CNT100;
   1:  PR[91] = PR[90];
   1:  PR[91,1] = PR[90,1] + -63.664;
   1:  PR[91,2] = PR[90,2] + 20.177;
   1:  PR[91,3] = PR[90,3] + 53.495;
   1:L PR[91] R[100]mm/sec CNT100;
   1:  PR[91,1] = PR[90,1] + -64.405;
   1:  PR[91,2] = PR[90,2] + 20.007;
   1:  PR[91,3] = PR[90,3] + 52.206;
   1:L PR[91] R[100]mm/sec CNT100;
   1:  PR[91,1] = PR[90,1] + -68.903;
   1:  PR[91,2] = PR[90,2] + 18.902;
   1:  PR[91,3] = PR[90,3] + 52.208;
   1:L PR[91] R[100]mm/sec CNT100;
   1:  PR[91,1] = PR[90,1] + -73.324;
   1:  PR[91,2] = PR[90,2] + 16.896;
   1:  PR[91,3] = PR[90,3] + 52.223;
   1:L PR[91] R[100]mm/sec CNT100;
   1:  PR[91,1] = PR[90,1] + -77.149;
   1:  PR[91,2] = PR[90,2] + 14.207;
   1:  PR[91,3] = PR[90,3] + 52.239;
   1:L PR[91] R[100]mm/sec CNT100;
   1:  PR[91,1] = PR[90,1] + -79.153;
   1:  PR[91,2] = PR[90,2] + 12.115;
   1:  PR[91,3] = PR[90,3] + 52.253;
   1:L PR[91] R[100]mm/sec CNT100;
   1:  PR[91,1] = PR[90,1] + -80.238;
   1:  PR[91,2] = PR[90,2] + 10.967;
   1:  PR[91,3] = PR[90,3] + 52.263;
   1:L PR[91] R[100]mm/sec CNT100;
   1:  PR[91,1] = PR[90,1] + -82.511;
   1:  PR[91,2] = PR[90,2] + 7.299;
   1:  PR[91,3] = PR[90,3] + 52.268;
   1:L PR[91] R[100]mm/sec CNT100;
   1:  PR[91,1] = PR[90,1] + -83.896;
   1:  PR[91,2] = PR[90,2] + 3.353;
   1:  PR[91,3] = PR[90,3] + 52.282;
   1:L PR[91] R[100]mm/sec CNT100;
   1:  PR[91,1] = PR[90,1] + -84.340;
   1:  PR[91,2] = PR[90,2] + -0.508;
   1:  PR[91,3] = PR[90,3] + 52.295;
   1:L PR[91] R[100]mm/sec CNT100;
   1:  PR[91,1] = PR[90,1] + -84.375;
   1:  PR[91,2] = PR[90,2] + -0.698;
   1:  PR[91,3] = PR[90,3] + 52.307;
   1:L PR[91] R[100]mm/sec CNT100;
   1:  PR[91,1] = PR[90,1] + -84.158;
   1:  PR[91,2] = PR[90,2] + -1.700;
   1:  PR[91,3] = PR[90,3] + 52.308;
   1:L PR[91] R[100]mm/sec CNT100;
   1:  PR[91,1] = PR[90,1] + -83.814;
   1:  PR[91,2] = PR[90,2] + -4.825;
   1:  PR[91,3] = PR[90,3] + 52.311;
   1:L PR[91] R[100]mm/sec CNT100;
   1:  PR[91,1] = PR[90,1] + -83.497;
   1:  PR[91,2] = PR[90,2] + -5.747;
   1:  PR[91,3] = PR[90,3] + 52.321;
   1:L PR[91] R[100]mm/sec CNT100;
   1:  PR[91,1] = PR[90,1] + -82.468;
   1:  PR[91,2] = PR[90,2] + -8.781;
   1:  PR[91,3] = PR[90,3] + 52.324;
   1:L PR[91] R[100]mm/sec CNT100;
   1:  PR[91,1] = PR[90,1] + -80.265;
   1:  PR[91,2] = PR[90,2] + -12.442;
   1:  PR[91,3] = PR[90,3] + 52.335;
   1:L PR[91] R[100]mm/sec CNT100;
   1:  PR[91,1] = PR[90,1] + -77.290;
   1:  PR[91,2] = PR[90,2] + -15.655;
   1:  PR[91,3] = PR[90,3] + 52.348;
   1:L PR[91] R[100]mm/sec CNT100;
   1:  PR[91,1] = PR[90,1] + -73.773;
   1:  PR[91,2] = PR[90,2] + -18.074;
   1:  PR[91,3] = PR[90,3] + 52.362;
   1:L PR[91] R[100]mm/sec CNT100;
   1:  PR[91,1] = PR[90,1] + -73.148;
   1:  PR[91,2] = PR[90,2] + -18.464;
   1:  PR[91,3] = PR[90,3] + 52.376;
   1:L PR[91] R[100]mm/sec CNT100;
   1:  PR[91,1] = PR[90,1] + -69.914;
   1:  PR[91,2] = PR[90,2] + -19.899;
   1:  PR[91,3] = PR[90,3] + 52.378;
   1:L PR[91] R[100]mm/sec CNT100;
   1:  PR[91,1] = PR[90,1] + -68.020;
   1:  PR[91,2] = PR[90,2] + -20.618;
   1:  PR[91,3] = PR[90,3] + 52.389;
   1:L PR[91] R[100]mm/sec CNT100;
   1:  PR[91,1] = PR[90,1] + -65.688;
   1:  PR[91,2] = PR[90,2] + -21.189;
   1:  PR[91,3] = PR[90,3] + 52.396;
   1:L PR[91] R[100]mm/sec CNT100;
   1:  PR[91,1] = PR[90,1] + -62.026;
   1:  PR[91,2] = PR[90,2] + -21.842;
   1:  PR[91,3] = PR[90,3] + 52.404;
   1:L PR[91] R[100]mm/sec CNT100;
   1:  PR[91,1] = PR[90,1] + -61.171;
   1:  PR[91,2] = PR[90,2] + -21.899;
   1:  PR[91,3] = PR[90,3] + 52.415;
   1:L PR[91] R[100]mm/sec CNT100;
   1:  PR[91,1] = PR[90,1] + -58.421;
   1:  PR[91,2] = PR[90,2] + -21.875;
   1:  PR[91,3] = PR[90,3] + 52.418;
   1:L PR[91] R[100]mm/sec CNT100;
   1:  PR[91,1] = PR[90,1] + -55.610;
   1:  PR[91,2] = PR[90,2] + -21.908;
   1:  PR[91,3] = PR[90,3] + 52.427;
   1:L PR[91] R[100]mm/sec CNT100;
   1:  PR[91,1] = PR[90,1] + -53.361;
   1:  PR[91,2] = PR[90,2] + -21.572;
   1:  PR[91,3] = PR[90,3] + 52.436;
   1:L PR[91] R[100]mm/sec CNT100;
   1:  PR[91,1] = PR[90,1] + -49.366;
   1:  PR[91,2] = PR[90,2] + -20.935;
   1:  PR[91,3] = PR[90,3] + 52.443;
   1:L PR[91] R[100]mm/sec CNT100;
   1:  PR[91,1] = PR[90,1] + -44.869;
   1:  PR[91,2] = PR[90,2] + -19.402;
   1:  PR[91,3] = PR[90,3] + 52.456;
   1:L PR[91] R[100]mm/sec CNT100;
   1:  PR[91,1] = PR[90,1] + -43.470;
   1:  PR[91,2] = PR[90,2] + -19.014;
   1:  PR[91,3] = PR[90,3] + 52.471;
   1:L PR[91] R[100]mm/sec CNT100;
   1:  PR[91,1] = PR[90,1] + -42.618;
   1:  PR[91,2] = PR[90,2] + -18.706;
   1:  PR[91,3] = PR[90,3] + 52.476;
   1:L PR[91] R[100]mm/sec CNT100;
   1:  PR[91,1] = PR[90,1] + -39.092;
   1:  PR[91,2] = PR[90,2] + -16.987;
   1:  PR[91,3] = PR[90,3] + 52.479;
   1:L PR[91] R[100]mm/sec CNT100;
   1:  PR[91,1] = PR[90,1] + -35.433;
   1:  PR[91,2] = PR[90,2] + -14.847;
   1:  PR[91,3] = PR[90,3] + 52.491;
   1:L PR[91] R[100]mm/sec CNT100;
   1:  PR[91,1] = PR[90,1] + -33.833;
   1:  PR[91,2] = PR[90,2] + -13.577;
   1:  PR[91,3] = PR[90,3] + 52.505;
   1:L PR[91] R[100]mm/sec CNT100;
   1:  PR[91,1] = PR[90,1] + -32.403;
   1:  PR[91,2] = PR[90,2] + -15.120;
   1:  PR[91,3] = PR[90,3] + 52.511;
   1:L PR[91] R[100]mm/sec CNT100;
   1:  PR[91,1] = PR[90,1] + -31.919;
   1:  PR[91,2] = PR[90,2] + -15.590;
   1:  PR[91,3] = PR[90,3] + 52.518;
   1:L PR[91] R[100]mm/sec CNT100;
   1:  PR[91,1] = PR[90,1] + -30.396;
   1:  PR[91,2] = PR[90,2] + -16.855;
   1:  PR[91,3] = PR[90,3] + 52.520;
   1:L PR[91] R[100]mm/sec CNT100;
   1:  PR[91,1] = PR[90,1] + -28.256;
   1:  PR[91,2] = PR[90,2] + -18.369;
   1:  PR[91,3] = PR[90,3] + 52.527;
   1:L PR[91] R[100]mm/sec CNT100;
   1:  PR[91,1] = PR[90,1] + -27.944;
   1:  PR[91,2] = PR[90,2] + -18.574;
   1:  PR[91,3] = PR[90,3] + 52.535;
   1:L PR[91] R[100]mm/sec CNT100;
   1:  PR[91,1] = PR[90,1] + -25.646;
   1:  PR[91,2] = PR[90,2] + -19.813;
   1:  PR[91,3] = PR[90,3] + 52.536;
   1:L PR[91] R[100]mm/sec CNT100;
   1:  PR[91,1] = PR[90,1] + -23.648;
   1:  PR[91,2] = PR[90,2] + -20.670;
   1:  PR[91,3] = PR[90,3] + 52.544;
   1:L PR[91] R[100]mm/sec CNT100;
   1:  PR[91,1] = PR[90,1] + -20.393;
   1:  PR[91,2] = PR[90,2] + -21.611;
   1:  PR[91,3] = PR[90,3] + 52.551;
   1:L PR[91] R[100]mm/sec CNT100;
   1:  PR[91,1] = PR[90,1] + -18.996;
   1:  PR[91,2] = PR[90,2] + -21.891;
   1:  PR[91,3] = PR[90,3] + 52.562;
   1:L PR[91] R[100]mm/sec CNT100;
   1:  PR[91,1] = PR[90,1] + -14.629;
   1:  PR[91,2] = PR[90,2] + -22.199;
   1:  PR[91,3] = PR[90,3] + 52.567;
   1:L PR[91] R[100]mm/sec CNT100;
   1:  PR[91,1] = PR[90,1] + -14.108;
   1:  PR[91,2] = PR[90,2] + -22.194;
   1:  PR[91,3] = PR[90,3] + 52.581;
   1:L PR[91] R[100]mm/sec CNT100;
   1:  PR[91,1] = PR[90,1] + -10.298;
   1:  PR[91,2] = PR[90,2] + -21.648;
   1:  PR[91,3] = PR[90,3] + 52.582;
   1:L PR[91] R[100]mm/sec CNT100;
   1:  PR[91,1] = PR[90,1] + -8.914;
   1:  PR[91,2] = PR[90,2] + -21.477;
   1:  PR[91,3] = PR[90,3] + 52.595;
   1:L PR[91] R[100]mm/sec CNT100;
   1:  PR[91,1] = PR[90,1] + -3.731;
   1:  PR[91,2] = PR[90,2] + -19.700;
   1:  PR[91,3] = PR[90,3] + 52.599;
   1:L PR[91] R[100]mm/sec CNT100;
   1:  PR[91,1] = PR[90,1] + -2.290;
   1:  PR[91,2] = PR[90,2] + -18.871;
   1:  PR[91,3] = PR[90,3] + 52.617;
   1:L PR[91] R[100]mm/sec CNT100;
   1:  PR[91,1] = PR[90,1] + 0.808;
   1:  PR[91,2] = PR[90,2] + -16.971;
   1:  PR[91,3] = PR[90,3] + 52.622;
   1:L PR[91] R[100]mm/sec CNT100;
   1:  PR[91,1] = PR[90,1] + 3.899;
   1:  PR[91,2] = PR[90,2] + -14.104;
   1:  PR[91,3] = PR[90,3] + 52.633;
   1:L PR[91] R[100]mm/sec CNT100;
   1:  PR[91,1] = PR[90,1] + 7.835;
   1:  PR[91,2] = PR[90,2] + -18.007;
   1:  PR[91,3] = PR[90,3] + 52.647;
   1:L PR[91] R[100]mm/sec CNT100;
   1:  PR[91,1] = PR[90,1] + 8.015;
   1:  PR[91,2] = PR[90,2] + -18.166;
   1:  PR[91,3] = PR[90,3] + 52.665;
   1:L PR[91] R[100]mm/sec CNT100;
   1:  PR[91,1] = PR[90,1] + 8.271;
   1:  PR[91,2] = PR[90,2] + -18.366;
   1:L PR[91] R[100]mm/sec CNT100;
   1:  PR[91,1] = PR[90,1] + 12.382;
   1:  PR[91,2] = PR[90,2] + -20.909;
   1:  PR[91,3] = PR[90,3] + 52.666;
   1:L PR[91] R[100]mm/sec CNT100;
   1:  PR[91,1] = PR[90,1] + 13.077;
   1:  PR[91,2] = PR[90,2] + -21.285;
   1:  PR[91,3] = PR[90,3] + 52.682;
   1:L PR[91] R[100]mm/sec CNT100;
   1:  PR[91,1] = PR[90,1] + 17.886;
   1:  PR[91,2] = PR[90,2] + -22.790;
   1:  PR[91,3] = PR[90,3] + 52.684;
   1:L PR[91] R[100]mm/sec CNT100;
   1:  PR[91,1] = PR[90,1] + 18.405;
   1:  PR[91,2] = PR[90,2] + -22.931;
   1:  PR[91,3] = PR[90,3] + 52.700;
   1:L PR[91] R[100]mm/sec CNT100;
   1:  PR[91,1] = PR[90,1] + 24.016;
   1:  PR[91,2] = PR[90,2] + -23.233;
   1:  PR[91,3] = PR[90,3] + 52.702;
   1:L PR[91] R[100]mm/sec CNT100;
   1:  PR[91,1] = PR[90,1] + 29.612;
   1:  PR[91,2] = PR[90,2] + -22.143;
   1:  PR[91,3] = PR[90,3] + 52.720;
   1:L PR[91] R[100]mm/sec CNT100;
   1:  PR[91,1] = PR[90,1] + 29.619;
   1:  PR[91,2] = PR[90,2] + -22.141;
   1:  PR[91,3] = PR[90,3] + 52.738;
   1:L PR[91] R[100]mm/sec CNT100;
   1:  PR[91,1] = PR[90,1] + 32.292;
   1:  PR[91,2] = PR[90,2] + -20.899;
   1:L PR[91] R[100]mm/sec CNT100;
   1:  PR[91,1] = PR[90,1] + 35.523;
   1:  PR[91,2] = PR[90,2] + -19.356;
   1:  PR[91,3] = PR[90,3] + 52.748;
   1:L PR[91] R[100]mm/sec CNT100;
   1:  PR[91,1] = PR[90,1] + 37.278;
   1:  PR[91,2] = PR[90,2] + -20.128;
   1:  PR[91,3] = PR[90,3] + 52.759;
   1:L PR[91] R[100]mm/sec CNT100;
   1:  PR[91,1] = PR[90,1] + 39.983;
   1:  PR[91,2] = PR[90,2] + -21.191;
   1:  PR[91,3] = PR[90,3] + 52.765;
   1:L PR[91] R[100]mm/sec CNT100;
   1:  PR[91,1] = PR[90,1] + 42.056;
   1:  PR[91,2] = PR[90,2] + -21.807;
   1:  PR[91,3] = PR[90,3] + 52.775;
   1:L PR[91] R[100]mm/sec CNT100;
   1:  PR[91,1] = PR[90,1] + 44.404;
   1:  PR[91,2] = PR[90,2] + -22.578;
   1:  PR[91,3] = PR[90,3] + 52.781;
   1:L PR[91] R[100]mm/sec CNT100;
   1:  PR[91,1] = PR[90,1] + 51.294;
   1:  PR[91,2] = PR[90,2] + -23.796;
   1:  PR[91,3] = PR[90,3] + 52.789;
   1:L PR[91] R[100]mm/sec CNT100;
   1:  PR[91,1] = PR[90,1] + 51.618;
   1:  PR[91,2] = PR[90,2] + -23.815;
   1:  PR[91,3] = PR[90,3] + 52.812;
   1:L PR[91] R[100]mm/sec CNT100;
   1:  PR[91,1] = PR[90,1] + 56.644;
   1:  PR[91,2] = PR[90,2] + -23.895;
   1:  PR[91,3] = PR[90,3] + 52.813;
   1:L PR[91] R[100]mm/sec CNT100;
   1:  PR[91,1] = PR[90,1] + 58.930;
   1:  PR[91,2] = PR[90,2] + -23.898;
   1:  PR[91,3] = PR[90,3] + 52.829;
   1:L PR[91] R[100]mm/sec CNT100;
   1:  PR[91,1] = PR[90,1] + 61.262;
   1:  PR[91,2] = PR[90,2] + -23.523;
   1:  PR[91,3] = PR[90,3] + 52.836;
   1:L PR[91] R[100]mm/sec CNT100;
   1:  PR[91,1] = PR[90,1] + 65.848;
   1:  PR[91,2] = PR[90,2] + -22.722;
   1:  PR[91,3] = PR[90,3] + 52.844;
   1:L PR[91] R[100]mm/sec CNT100;
   1:  PR[91,1] = PR[90,1] + 70.897;
   1:  PR[91,2] = PR[90,2] + -20.821;
   1:  PR[91,3] = PR[90,3] + 52.858;
   1:L PR[91] R[100]mm/sec CNT100;
   1:  PR[91,1] = PR[90,1] + 72.535;
   1:  PR[91,2] = PR[90,2] + -19.930;
   1:  PR[91,3] = PR[90,3] + 52.876;
   1:L PR[91] R[100]mm/sec CNT100;
   1:  PR[91,1] = PR[90,1] + 75.419;
   1:  PR[91,2] = PR[90,2] + -18.127;
   1:  PR[91,3] = PR[90,3] + 52.882;
   1:L PR[91] R[100]mm/sec CNT100;
   1:  PR[91,1] = PR[90,1] + 78.058;
   1:  PR[91,2] = PR[90,2] + -15.842;
   1:  PR[91,3] = PR[90,3] + 52.892;
   1:L PR[91] R[100]mm/sec CNT100;
   1:  PR[91,1] = PR[90,1] + 79.327;
   1:  PR[91,2] = PR[90,2] + -14.624;
   1:  PR[91,3] = PR[90,3] + 52.904;
   1:L PR[91] R[100]mm/sec CNT100;
   1:  PR[91,1] = PR[90,1] + 81.972;
   1:  PR[91,2] = PR[90,2] + -10.980;
   1:  PR[91,3] = PR[90,3] + 52.909;
   1:L PR[91] R[100]mm/sec CNT100;
   1:  PR[91,1] = PR[90,1] + 82.342;
   1:  PR[91,2] = PR[90,2] + -10.424;
   1:  PR[91,3] = PR[90,3] + 52.924;
   1:L PR[91] R[100]mm/sec CNT100;
   1:  PR[91,1] = PR[90,1] + 84.250;
   1:  PR[91,2] = PR[90,2] + -5.685;
   1:  PR[91,3] = PR[90,3] + 52.926;
   1:L PR[91] R[100]mm/sec CNT100;
   1:  PR[91,1] = PR[90,1] + 84.909;
   1:  PR[91,2] = PR[90,2] + -0.727;
   1:  PR[91,3] = PR[90,3] + 52.942;
   1:L PR[91] R[100]mm/sec CNT100;
   1:  PR[91,1] = PR[90,1] + 84.313;
   1:  PR[91,2] = PR[90,2] + 3.861;
   1:  PR[91,3] = PR[90,3] + 52.958;
   1:L PR[91] R[100]mm/sec CNT100;
   1:  PR[91,1] = PR[90,1] + 84.256;
   1:  PR[91,2] = PR[90,2] + 4.148;
   1:  PR[91,3] = PR[90,3] + 52.973;
   1:L PR[91] R[100]mm/sec CNT100;
   1:  PR[91,1] = PR[90,1] + 84.245;
   1:  PR[91,2] = PR[90,2] + 4.240;
   1:  PR[91,3] = PR[90,3] + 52.974;
   1:L PR[91] R[100]mm/sec CNT100;
   1:  PR[91,1] = PR[90,1] + 82.342;
   1:  PR[91,2] = PR[90,2] + 8.966;
   1:L PR[91] R[100]mm/sec CNT100;
   1:  PR[91,1] = PR[90,1] + 81.969;
   1:  PR[91,2] = PR[90,2] + 9.524;
   1:  PR[91,3] = PR[90,3] + 52.990;
   1:L PR[91] R[100]mm/sec CNT100;
   1:  PR[91,1] = PR[90,1] + 79.323;
   1:  PR[91,2] = PR[90,2] + 13.170;
   1:  PR[91,3] = PR[90,3] + 52.992;
   1:L PR[91] R[100]mm/sec CNT100;
   1:  PR[91,1] = PR[90,1] + 78.046;
   1:  PR[91,2] = PR[90,2] + 14.393;
   1:  PR[91,3] = PR[90,3] + 53.007;
   1:L PR[91] R[100]mm/sec CNT100;
   1:  PR[91,1] = PR[90,1] + 75.406;
   1:  PR[91,2] = PR[90,2] + 16.677;
   1:  PR[91,3] = PR[90,3] + 53.012;
   1:L PR[91] R[100]mm/sec CNT100;
   1:  PR[91,1] = PR[90,1] + 72.500;
   1:  PR[91,2] = PR[90,2] + 18.489;
   1:  PR[91,3] = PR[90,3] + 53.024;
   1:L PR[91] R[100]mm/sec CNT100;
   1:  PR[91,1] = PR[90,1] + 70.869;
   1:  PR[91,2] = PR[90,2] + 19.376;
   1:  PR[91,3] = PR[90,3] + 53.035;
   1:L PR[91] R[100]mm/sec CNT100;
   1:  PR[91,1] = PR[90,1] + 65.788;
   1:  PR[91,2] = PR[90,2] + 21.279;
   1:  PR[91,3] = PR[90,3] + 53.040;
   1:L PR[91] R[100]mm/sec CNT100;
   1:  PR[91,1] = PR[90,1] + 61.230;
   1:  PR[91,2] = PR[90,2] + 22.064;
   1:  PR[91,3] = PR[90,3] + 53.058;
   1:L PR[91] R[100]mm/sec CNT100;
   1:  PR[91,1] = PR[90,1] + 58.908;
   1:  PR[91,2] = PR[90,2] + 22.441;
   1:  PR[91,3] = PR[90,3] + 53.073;
   1:L PR[91] R[100]mm/sec CNT100;
   1:  PR[91,1] = PR[90,1] + 56.639;
   1:  PR[91,2] = PR[90,2] + 22.431;
   1:  PR[91,3] = PR[90,3] + 53.080;
   1:L PR[91] R[100]mm/sec CNT100;
   1:  PR[91,1] = PR[90,1] + 51.644;
   1:  PR[91,2] = PR[90,2] + 22.359;
   1:  PR[91,3] = PR[90,3] + 53.087;
   1:L PR[91] R[100]mm/sec CNT100;
   1:  PR[91,1] = PR[90,1] + 51.339;
   1:  PR[91,2] = PR[90,2] + 22.342;
   1:  PR[91,3] = PR[90,3] + 53.103;
   1:L PR[91] R[100]mm/sec CNT100;
   1:  PR[91,1] = PR[90,1] + 46.971;
   1:  PR[91,2] = PR[90,2] + 21.551;
   1:  PR[91,3] = PR[90,3] + 53.104;
   1:L PR[91] R[100]mm/sec CNT100;
   1:  PR[91,1] = PR[90,1] + 44.406;
   1:  PR[91,2] = PR[90,2] + 21.119;
   1:  PR[91,3] = PR[90,3] + 53.118;
   1:L PR[91] R[100]mm/sec CNT100;
   1:  PR[91,1] = PR[90,1] + 42.056;
   1:  PR[91,2] = PR[90,2] + 20.348;
   1:  PR[91,3] = PR[90,3] + 53.127;
   1:L PR[91] R[100]mm/sec CNT100;
   1:  PR[91,1] = PR[90,1] + 39.983;
   1:  PR[91,2] = PR[90,2] + 19.732;
   1:  PR[91,3] = PR[90,3] + 53.135;
   1:L PR[91] R[100]mm/sec CNT100;
   1:  PR[91,1] = PR[90,1] + 37.277;
   1:  PR[91,2] = PR[90,2] + 18.669;
   1:  PR[91,3] = PR[90,3] + 53.141;
   1:L PR[91] R[100]mm/sec CNT100;
   1:  PR[91,1] = PR[90,1] + 35.523;
   1:  PR[91,2] = PR[90,2] + 17.898;
   1:  PR[91,3] = PR[90,3] + 53.151;
   1:L PR[91] R[100]mm/sec CNT100;
   1:  PR[91,1] = PR[90,1] + 32.292;
   1:  PR[91,2] = PR[90,2] + 19.440;
   1:  PR[91,3] = PR[90,3] + 53.157;
   1:L PR[91] R[100]mm/sec CNT100;
   1:  PR[91,1] = PR[90,1] + 29.617;
   1:  PR[91,2] = PR[90,2] + 20.683;
   1:  PR[91,3] = PR[90,3] + 53.168;
   1:L PR[91] R[100]mm/sec CNT100;
   1:  PR[91,1] = PR[90,1] + 24.273;
   1:  PR[91,2] = PR[90,2] + 21.729;
   1:  PR[91,3] = PR[90,3] + 53.178;
   1:L PR[91] R[100]mm/sec CNT100;
   1:  PR[91,1] = PR[90,1] + 24.028;
   1:  PR[91,2] = PR[90,2] + 21.775;
   1:  PR[91,3] = PR[90,3] + 53.195;
   1:L PR[91] R[100]mm/sec CNT100;
   1:  PR[91,1] = PR[90,1] + 18.412;
   1:  PR[91,2] = PR[90,2] + 21.474;
   1:  PR[91,3] = PR[90,3] + 53.196;
   1:L PR[91] R[100]mm/sec CNT100;
   1:  PR[91,1] = PR[90,1] + 17.893;
   1:  PR[91,2] = PR[90,2] + 21.332;
   1:  PR[91,3] = PR[90,3] + 53.214;
   1:L PR[91] R[100]mm/sec CNT100;
   1:  PR[91,1] = PR[90,1] + 13.085;
   1:  PR[91,2] = PR[90,2] + 19.830;
   1:  PR[91,3] = PR[90,3] + 53.216;
   1:L PR[91] R[100]mm/sec CNT100;
   1:  PR[91,1] = PR[90,1] + 12.386;
   1:  PR[91,2] = PR[90,2] + 19.451;
   1:  PR[91,3] = PR[90,3] + 53.232;
   1:L PR[91] R[100]mm/sec CNT100;
   1:  PR[91,1] = PR[90,1] + 8.298;
   1:  PR[91,2] = PR[90,2] + 16.925;
   1:  PR[91,3] = PR[90,3] + 53.234;
   1:L PR[91] R[100]mm/sec CNT100;
   1:  PR[91,1] = PR[90,1] + 7.780;
   1:  PR[91,2] = PR[90,2] + 16.498;
   1:  PR[91,3] = PR[90,3] + 53.249;
   1:L PR[91] R[100]mm/sec CNT100;
   1:  PR[91,1] = PR[90,1] + 7.368;
   1:  PR[91,2] = PR[90,2] + 16.113;
   1:  PR[91,3] = PR[90,3] + 53.252;
   1:L PR[91] R[100]mm/sec CNT100;
   1:  PR[91,1] = PR[90,1] + 3.909;
   1:  PR[91,2] = PR[90,2] + 12.520;
   1:  PR[91,3] = PR[90,3] + 53.253;
   1:L PR[91] R[100]mm/sec CNT100;
   1:  PR[91,1] = PR[90,1] + 1.090;
   1:  PR[91,2] = PR[90,2] + 15.271;
   1:  PR[91,3] = PR[90,3] + 53.269;
   1:L PR[91] R[100]mm/sec CNT100;
   1:  PR[91,1] = PR[90,1] + 0.857;
   1:  PR[91,2] = PR[90,2] + 15.476;
   1:  PR[91,3] = PR[90,3] + 53.282;
   1:L PR[91] R[100]mm/sec CNT100;
   1:  PR[91,1] = PR[90,1] + -2.238;
   1:  PR[91,2] = PR[90,2] + 17.381;
   1:  PR[91,3] = PR[90,3] + 53.283;
   1:L PR[91] R[100]mm/sec CNT100;
   1:  PR[91,1] = PR[90,1] + -3.706;
   1:  PR[91,2] = PR[90,2] + 18.229;
   1:  PR[91,3] = PR[90,3] + 53.295;
   1:L PR[91] R[100]mm/sec CNT100;
   1:  PR[91,1] = PR[90,1] + -8.881;
   1:  PR[91,2] = PR[90,2] + 20.010;
   1:  PR[91,3] = PR[90,3] + 53.300;
   1:L PR[91] R[100]mm/sec CNT100;
   1:  PR[91,1] = PR[90,1] + -10.300;
   1:  PR[91,2] = PR[90,2] + 20.188;
   1:  PR[91,3] = PR[90,3] + 53.317;
   1:L PR[91] R[100]mm/sec CNT100;
   1:  PR[91,1] = PR[90,1] + -14.076;
   1:  PR[91,2] = PR[90,2] + 20.734;
   1:  PR[91,3] = PR[90,3] + 53.322;
   1:L PR[91] R[100]mm/sec CNT100;
   1:  PR[91,1] = PR[90,1] + -14.592;
   1:  PR[91,2] = PR[90,2] + 20.739;
   1:  PR[91,3] = PR[90,3] + 53.334;
   1:L PR[91] R[100]mm/sec CNT100;
   1:  PR[91,1] = PR[90,1] + -18.967;
   1:  PR[91,2] = PR[90,2] + 20.437;
   1:  PR[91,3] = PR[90,3] + 53.336;
   1:L PR[91] R[100]mm/sec CNT100;
   1:  PR[91,1] = PR[90,1] + -20.360;
   1:  PR[91,2] = PR[90,2] + 20.158;
   1:  PR[91,3] = PR[90,3] + 53.350;
   1:L PR[91] R[100]mm/sec CNT100;
   1:  PR[91,1] = PR[90,1] + -23.623;
   1:  PR[91,2] = PR[90,2] + 19.221;
   1:  PR[91,3] = PR[90,3] + 53.354;
   1:L PR[91] R[100]mm/sec CNT100;
   1:  PR[91,1] = PR[90,1] + -25.620;
   1:  PR[91,2] = PR[90,2] + 18.365;
   1:  PR[91,3] = PR[90,3] + 53.365;
   1:L PR[91] R[100]mm/sec CNT100;
   1:  PR[91,1] = PR[90,1] + -27.873;
   1:  PR[91,2] = PR[90,2] + 17.158;
   1:  PR[91,3] = PR[90,3] + 53.372;
   1:L PR[91] R[100]mm/sec CNT100;
   1:  PR[91,1] = PR[90,1] + -30.316;
   1:  PR[91,2] = PR[90,2] + 15.446;
   1:  PR[91,3] = PR[90,3] + 53.380;
   1:L PR[91] R[100]mm/sec CNT100;
   1:  PR[91,1] = PR[90,1] + -31.003;
   1:  PR[91,2] = PR[90,2] + 14.947;
   1:  PR[91,3] = PR[90,3] + 53.390;
   1:L PR[91] R[100]mm/sec CNT100;
   1:  PR[91,1] = PR[90,1] + -31.735;
   1:  PR[91,2] = PR[90,2] + 14.304;
   1:  PR[91,3] = PR[90,3] + 53.392;
   1:L PR[91] R[100]mm/sec CNT100;
   1:  PR[91,1] = PR[90,1] + -33.805;
   1:  PR[91,2] = PR[90,2] + 12.267;
   1:  PR[91,3] = PR[90,3] + 53.396;
   1:L PR[91] R[100]mm/sec CNT100;
   1:  PR[91,1] = PR[90,1] + -37.015;
   1:  PR[91,2] = PR[90,2] + 14.429;
   1:  PR[91,3] = PR[90,3] + 53.405;
   1:L PR[91] R[100]mm/sec CNT100;
   1:  PR[91,1] = PR[90,1] + -39.167;
   1:  PR[91,2] = PR[90,2] + 15.560;
   1:  PR[91,3] = PR[90,3] + 53.417;
   1:L PR[91] R[100]mm/sec CNT100;
   1:  PR[91,1] = PR[90,1] + -41.600;
   1:  PR[91,2] = PR[90,2] + 16.570;
   1:  PR[91,3] = PR[90,3] + 53.425;
   1:L PR[91] R[100]mm/sec CNT100;
   1:  PR[91,1] = PR[90,1] + -43.569;
   1:  PR[91,2] = PR[90,2] + 17.552;
   1:  PR[91,3] = PR[90,3] + 53.433;
   1:L PR[91] R[100]mm/sec CNT100;
   1:  PR[91,1] = PR[90,1] + -44.607;
   1:  PR[91,2] = PR[90,2] + 18.033;
   1:  PR[91,3] = PR[90,3] + 53.440;
   1:L PR[91] R[100]mm/sec CNT100;
   1:  PR[91,1] = PR[90,1] + -47.534;
   1:  PR[91,2] = PR[90,2] + 18.865;
   1:  PR[91,3] = PR[90,3] + 53.444;
   1:L PR[91] R[100]mm/sec CNT100;
   1:  PR[91,1] = PR[90,1] + -51.386;
   1:  PR[91,2] = PR[90,2] + 19.873;
   1:  PR[91,3] = PR[90,3] + 53.454;
   1:L PR[91] R[100]mm/sec CNT100;
   1:  PR[91,1] = PR[90,1] + -52.453;
   1:  PR[91,2] = PR[90,2] + 19.978;
   1:  PR[91,3] = PR[90,3] + 53.466;
   1:L PR[91] R[100]mm/sec CNT100;
   1:  PR[91,1] = PR[90,1] + -56.156;
   1:  PR[91,2] = PR[90,2] + 20.410;
   1:  PR[91,3] = PR[90,3] + 53.470;
   1:L PR[91] R[100]mm/sec CNT100;
   1:  PR[91,1] = PR[90,1] + -57.715;
   1:  PR[91,2] = PR[90,2] + 20.561;
   1:  PR[91,3] = PR[90,3] + 53.482;
   1:L PR[91] R[100]mm/sec CNT100;
   1:  PR[91,1] = PR[90,1] + -60.285;
   1:  PR[91,2] = PR[90,2] + 20.419;
   1:  PR[91,3] = PR[90,3] + 53.487;
   1:L PR[91] R[100]mm/sec CNT100;
   1:  PR[91] = PR[90];
   1:  PR[91,1] = PR[90,1] + -62.642;
   1:  PR[91,2] = PR[90,2] + 20.365;
   1:  PR[91,3] = PR[90,3] + 54.795;
   1:L PR[91] R[100]mm/sec CNT100;
   1:  PR[91,1] = PR[90,1] + -64.185;
   1:  PR[91,2] = PR[90,2] + 20.010;
   1:  PR[91,3] = PR[90,3] + 53.503;
   1:L PR[91] R[100]mm/sec CNT100;
   1:  PR[91,1] = PR[90,1] + -68.190;
   1:  PR[91,2] = PR[90,2] + 19.037;
   1:  PR[91,3] = PR[90,3] + 53.508;
   1:L PR[91] R[100]mm/sec CNT100;
   1:  PR[91,1] = PR[90,1] + -68.766;
   1:  PR[91,2] = PR[90,2] + 18.787;
   1:  PR[91,3] = PR[90,3] + 53.522;
   1:L PR[91] R[100]mm/sec CNT100;
   1:  PR[91,1] = PR[90,1] + -72.684;
   1:  PR[91,2] = PR[90,2] + 17.004;
   1:  PR[91,3] = PR[90,3] + 53.524;
   1:L PR[91] R[100]mm/sec CNT100;
   1:  PR[91,1] = PR[90,1] + -76.525;
   1:  PR[91,2] = PR[90,2] + 14.297;
   1:  PR[91,3] = PR[90,3] + 53.538;
   1:L PR[91] R[100]mm/sec CNT100;
   1:  PR[91,1] = PR[90,1] + -79.633;
   1:  PR[91,2] = PR[90,2] + 11.029;
   1:  PR[91,3] = PR[90,3] + 53.553;
   1:L PR[91] R[100]mm/sec CNT100;
   1:  PR[91,1] = PR[90,1] + -81.091;
   1:  PR[91,2] = PR[90,2] + 8.683;
   1:  PR[91,3] = PR[90,3] + 53.567;
   1:L PR[91] R[100]mm/sec CNT100;
   1:  PR[91,1] = PR[90,1] + -81.912;
   1:  PR[91,2] = PR[90,2] + 7.346;
   1:  PR[91,3] = PR[90,3] + 53.576;
   1:L PR[91] R[100]mm/sec CNT100;
   1:  PR[91,1] = PR[90,1] + -83.303;
   1:  PR[91,2] = PR[90,2] + 3.375;
   1:  PR[91,3] = PR[90,3] + 53.581;
   1:L PR[91] R[100]mm/sec CNT100;
   1:  PR[91,1] = PR[90,1] + -83.681;
   1:  PR[91,2] = PR[90,2] + 0.100;
   1:  PR[91,3] = PR[90,3] + 53.595;
   1:L PR[91] R[100]mm/sec CNT100;
   1:  PR[91,1] = PR[90,1] + -83.828;
   1:  PR[91,2] = PR[90,2] + -0.698;
   1:  PR[91,3] = PR[90,3] + 53.606;
   1:L PR[91] R[100]mm/sec CNT100;
   1:  PR[91,1] = PR[90,1] + -83.715;
   1:  PR[91,2] = PR[90,2] + -1.219;
   1:  PR[91,3] = PR[90,3] + 53.608;
   1:L PR[91] R[100]mm/sec CNT100;
   1:  PR[91,1] = PR[90,1] + -83.316;
   1:  PR[91,2] = PR[90,2] + -4.844;
   1:  PR[91,3] = PR[90,3] + 53.610;
   1:L PR[91] R[100]mm/sec CNT100;
   1:  PR[91,1] = PR[90,1] + -83.154;
   1:  PR[91,2] = PR[90,2] + -5.314;
   1:  PR[91,3] = PR[90,3] + 53.622;
   1:L PR[91] R[100]mm/sec CNT100;
   1:  PR[91,1] = PR[90,1] + -81.965;
   1:  PR[91,2] = PR[90,2] + -8.821;
   1:  PR[91,3] = PR[90,3] + 53.623;
   1:L PR[91] R[100]mm/sec CNT100;
   1:  PR[91,1] = PR[90,1] + -79.754;
   1:  PR[91,2] = PR[90,2] + -12.500;
   1:  PR[91,3] = PR[90,3] + 53.635;
   1:L PR[91] R[100]mm/sec CNT100;
   1:  PR[91,1] = PR[90,1] + -79.487;
   1:  PR[91,2] = PR[90,2] + -12.789;
   1:  PR[91,3] = PR[90,3] + 53.649;
   1:L PR[91] R[100]mm/sec CNT100;
   1:  PR[91,1] = PR[90,1] + -76.824;
   1:  PR[91,2] = PR[90,2] + -15.521;
   1:  PR[91,3] = PR[90,3] + 53.650;
   1:L PR[91] R[100]mm/sec CNT100;
   1:  PR[91,1] = PR[90,1] + -76.519;
   1:  PR[91,2] = PR[90,2] + -15.811;
   1:  PR[91,3] = PR[90,3] + 53.663;
   1:L PR[91] R[100]mm/sec CNT100;
   1:  PR[91,1] = PR[90,1] + -73.436;
   1:  PR[91,2] = PR[90,2] + -17.930;
   1:  PR[91,3] = PR[90,3] + 53.664;
   1:L PR[91] R[100]mm/sec CNT100;
   1:  PR[91,1] = PR[90,1] + -72.224;
   1:  PR[91,2] = PR[90,2] + -18.685;
   1:  PR[91,3] = PR[90,3] + 53.676;
   1:L PR[91] R[100]mm/sec CNT100;
   1:  PR[91,1] = PR[90,1] + -69.590;
   1:  PR[91,2] = PR[90,2] + -19.854;
   1:  PR[91,3] = PR[90,3] + 53.681;
   1:L PR[91] R[100]mm/sec CNT100;
   1:  PR[91,1] = PR[90,1] + -66.979;
   1:  PR[91,2] = PR[90,2] + -20.846;
   1:  PR[91,3] = PR[90,3] + 53.690;
   1:L PR[91] R[100]mm/sec CNT100;
   1:  PR[91,1] = PR[90,1] + -65.356;
   1:  PR[91,2] = PR[90,2] + -21.243;
   1:  PR[91,3] = PR[90,3] + 53.699;
   1:L PR[91] R[100]mm/sec CNT100;
   1:  PR[91,1] = PR[90,1] + -60.847;
   1:  PR[91,2] = PR[90,2] + -22.047;
   1:  PR[91,3] = PR[90,3] + 53.704;
   1:L PR[91] R[100]mm/sec CNT100;
   1:  PR[91,1] = PR[90,1] + -60.807;
   1:  PR[91,2] = PR[90,2] + -22.050;
   1:  PR[91,3] = PR[90,3] + 53.719;
   1:L PR[91] R[100]mm/sec CNT100;
   1:  PR[91,1] = PR[90,1] + -60.254;
   1:  PR[91,2] = PR[90,2] + -22.045;
   1:L PR[91] R[100]mm/sec CNT100;
   1:  PR[91,1] = PR[90,1] + -54.547;
   1:  PR[91,2] = PR[90,2] + -22.112;
   1:  PR[91,3] = PR[90,3] + 53.721;
   1:L PR[91] R[100]mm/sec CNT100;
   1:  PR[91,1] = PR[90,1] + -49.928;
   1:  PR[91,2] = PR[90,2] + -21.421;
   1:  PR[91,3] = PR[90,3] + 53.740;
   1:L PR[91] R[100]mm/sec CNT100;
   1:  PR[91,1] = PR[90,1] + -48.243;
   1:  PR[91,2] = PR[90,2] + -21.152;
   1:  PR[91,3] = PR[90,3] + 53.755;
   1:L PR[91] R[100]mm/sec CNT100;
   1:  PR[91,1] = PR[90,1] + -46.295;
   1:  PR[91,2] = PR[90,2] + -20.488;
   1:  PR[91,3] = PR[90,3] + 53.760;
   1:L PR[91] R[100]mm/sec CNT100;
   1:  PR[91,1] = PR[90,1] + -42.712;
   1:  PR[91,2] = PR[90,2] + -19.494;
   1:  PR[91,3] = PR[90,3] + 53.767;
   1:L PR[91] R[100]mm/sec CNT100;
   1:  PR[91,1] = PR[90,1] + -40.282;
   1:  PR[91,2] = PR[90,2] + -18.616;
   1:  PR[91,3] = PR[90,3] + 53.779;
   1:L PR[91] R[100]mm/sec CNT100;
   1:  PR[91,1] = PR[90,1] + -38.285;
   1:  PR[91,2] = PR[90,2] + -17.642;
   1:  PR[91,3] = PR[90,3] + 53.787;
   1:L PR[91] R[100]mm/sec CNT100;
   1:  PR[91,1] = PR[90,1] + -35.613;
   1:  PR[91,2] = PR[90,2] + -16.080;
   1:  PR[91,3] = PR[90,3] + 53.794;
   1:L PR[91] R[100]mm/sec CNT100;
   1:  PR[91,1] = PR[90,1] + -32.715;
   1:  PR[91,2] = PR[90,2] + -14.733;
   1:  PR[91,3] = PR[90,3] + 53.804;
   1:L PR[91] R[100]mm/sec CNT100;
   1:  PR[91,1] = PR[90,1] + -29.826;
   1:  PR[91,2] = PR[90,2] + -17.134;
   1:  PR[91,3] = PR[90,3] + 53.815;
   1:L PR[91] R[100]mm/sec CNT100;
   1:  PR[91,1] = PR[90,1] + -28.200;
   1:  PR[91,2] = PR[90,2] + -18.285;
   1:  PR[91,3] = PR[90,3] + 53.827;
   1:L PR[91] R[100]mm/sec CNT100;
   1:  PR[91,1] = PR[90,1] + -27.745;
   1:  PR[91,2] = PR[90,2] + -18.586;
   1:  PR[91,3] = PR[90,3] + 53.833;
   1:L PR[91] R[100]mm/sec CNT100;
   1:  PR[91,1] = PR[90,1] + -24.916;
   1:  PR[91,2] = PR[90,2] + -20.110;
   1:  PR[91,3] = PR[90,3] + 53.835;
   1:L PR[91] R[100]mm/sec CNT100;
   1:  PR[91,1] = PR[90,1] + -23.434;
   1:  PR[91,2] = PR[90,2] + -20.746;
   1:  PR[91,3] = PR[90,3] + 53.845;
   1:L PR[91] R[100]mm/sec CNT100;
   1:  PR[91,1] = PR[90,1] + -19.564;
   1:  PR[91,2] = PR[90,2] + -21.864;
   1:  PR[91,3] = PR[90,3] + 53.851;
   1:L PR[91] R[100]mm/sec CNT100;
   1:  PR[91,1] = PR[90,1] + -18.758;
   1:  PR[91,2] = PR[90,2] + -22.026;
   1:  PR[91,3] = PR[90,3] + 53.864;
   1:L PR[91] R[100]mm/sec CNT100;
   1:  PR[91,1] = PR[90,1] + -13.735;
   1:  PR[91,2] = PR[90,2] + -22.373;
   1:  PR[91,3] = PR[90,3] + 53.866;
   1:L PR[91] R[100]mm/sec CNT100;
   1:  PR[91,1] = PR[90,1] + -8.901;
   1:  PR[91,2] = PR[90,2] + -21.758;
   1:  PR[91,3] = PR[90,3] + 53.883;
   1:L PR[91] R[100]mm/sec CNT100;
   1:  PR[91,1] = PR[90,1] + -8.210;
   1:  PR[91,2] = PR[90,2] + -21.679;
   1:  PR[91,3] = PR[90,3] + 53.898;
   1:L PR[91] R[100]mm/sec CNT100;
   1:  PR[91,1] = PR[90,1] + -7.082;
   1:  PR[91,2] = PR[90,2] + -21.314;
   1:  PR[91,3] = PR[90,3] + 53.900;
   1:L PR[91] R[100]mm/sec CNT100;
   1:  PR[91,1] = PR[90,1] + -3.044;
   1:  PR[91,2] = PR[90,2] + -19.923;
   1:  PR[91,3] = PR[90,3] + 53.904;
   1:L PR[91] R[100]mm/sec CNT100;
   1:  PR[91,1] = PR[90,1] + -0.722;
   1:  PR[91,2] = PR[90,2] + -18.589;
   1:  PR[91,3] = PR[90,3] + 53.918;
   1:L PR[91] R[100]mm/sec CNT100;
   1:  PR[91,1] = PR[90,1] + 1.518;
   1:  PR[91,2] = PR[90,2] + -17.215;
   1:  PR[91,3] = PR[90,3] + 53.927;
   1:L PR[91] R[100]mm/sec CNT100;
   1:  PR[91,1] = PR[90,1] + 4.132;
   1:  PR[91,2] = PR[90,2] + -14.791;
   1:  PR[91,3] = PR[90,3] + 53.935;
   1:L PR[91] R[100]mm/sec CNT100;
   1:  PR[91,1] = PR[90,1] + 7.385;
   1:  PR[91,2] = PR[90,2] + -18.017;
   1:  PR[91,3] = PR[90,3] + 53.947;
   1:L PR[91] R[100]mm/sec CNT100;
   1:  PR[91,1] = PR[90,1] + 7.693;
   1:  PR[91,2] = PR[90,2] + -18.287;
   1:  PR[91,3] = PR[90,3] + 53.962;
   1:L PR[91] R[100]mm/sec CNT100;
   1:  PR[91,1] = PR[90,1] + 8.132;
   1:  PR[91,2] = PR[90,2] + -18.632;
   1:  PR[91,3] = PR[90,3] + 53.963;
   1:L PR[91] R[100]mm/sec CNT100;
   1:  PR[91,1] = PR[90,1] + 11.740;
   1:  PR[91,2] = PR[90,2] + -20.863;
   1:  PR[91,3] = PR[90,3] + 53.965;
   1:L PR[91] R[100]mm/sec CNT100;
   1:  PR[91,1] = PR[90,1] + 12.954;
   1:  PR[91,2] = PR[90,2] + -21.520;
   1:  PR[91,3] = PR[90,3] + 53.978;
   1:L PR[91] R[100]mm/sec CNT100;
   1:  PR[91,1] = PR[90,1] + 17.211;
   1:  PR[91,2] = PR[90,2] + -22.852;
   1:  PR[91,3] = PR[90,3] + 53.983;
   1:L PR[91] R[100]mm/sec CNT100;
   1:  PR[91,1] = PR[90,1] + 18.286;
   1:  PR[91,2] = PR[90,2] + -23.146;
   1:  PR[91,3] = PR[90,3] + 53.997;
   1:L PR[91] R[100]mm/sec CNT100;
   1:  PR[91,1] = PR[90,1] + 23.010;
   1:  PR[91,2] = PR[90,2] + -23.406;
   1:  PR[91,3] = PR[90,3] + 54.001;
   1:L PR[91] R[100]mm/sec CNT100;
   1:  PR[91,1] = PR[90,1] + 23.880;
   1:  PR[91,2] = PR[90,2] + -23.441;
   1:  PR[91,3] = PR[90,3] + 54.016;
   1:L PR[91] R[100]mm/sec CNT100;
   1:  PR[91,1] = PR[90,1] + 29.504;
   1:  PR[91,2] = PR[90,2] + -22.348;
   1:  PR[91,3] = PR[90,3] + 54.019;
   1:L PR[91] R[100]mm/sec CNT100;
   1:  PR[91,1] = PR[90,1] + 29.939;
   1:  PR[91,2] = PR[90,2] + -22.189;
   1:  PR[91,3] = PR[90,3] + 54.037;
   1:L PR[91] R[100]mm/sec CNT100;
   1:  PR[91,1] = PR[90,1] + 34.798;
   1:  PR[91,2] = PR[90,2] + -19.931;
   1:  PR[91,3] = PR[90,3] + 54.039;
   1:L PR[91] R[100]mm/sec CNT100;
   1:  PR[91,1] = PR[90,1] + 39.331;
   1:  PR[91,2] = PR[90,2] + -21.711;
   1:  PR[91,3] = PR[90,3] + 54.056;
   1:L PR[91] R[100]mm/sec CNT100;
   1:  PR[91,1] = PR[90,1] + 43.236;
   1:  PR[91,2] = PR[90,2] + -22.874;
   1:  PR[91,3] = PR[90,3] + 54.072;
   1:L PR[91] R[100]mm/sec CNT100;
   1:  PR[91,1] = PR[90,1] + 49.703;
   1:  PR[91,2] = PR[90,2] + -24.004;
   1:  PR[91,3] = PR[90,3] + 54.085;
   1:L PR[91] R[100]mm/sec CNT100;
   1:  PR[91,1] = PR[90,1] + 51.113;
   1:  PR[91,2] = PR[90,2] + -24.085;
   1:  PR[91,3] = PR[90,3] + 54.106;
   1:L PR[91] R[100]mm/sec CNT100;
   1:  PR[91,1] = PR[90,1] + 53.961;
   1:  PR[91,2] = PR[90,2] + -24.100;
   1:  PR[91,3] = PR[90,3] + 54.111;
   1:L PR[91] R[100]mm/sec CNT100;
   1:  PR[91,1] = PR[90,1] + 56.476;
   1:  PR[91,2] = PR[90,2] + -24.146;
   1:  PR[91,3] = PR[90,3] + 54.120;
   1:L PR[91] R[100]mm/sec CNT100;
   1:  PR[91,1] = PR[90,1] + 57.774;
   1:  PR[91,2] = PR[90,2] + -24.147;
   1:  PR[91,3] = PR[90,3] + 54.128;
   1:L PR[91] R[100]mm/sec CNT100;
   1:  PR[91,1] = PR[90,1] + 61.090;
   1:  PR[91,2] = PR[90,2] + -23.614;
   1:  PR[91,3] = PR[90,3] + 54.132;
   1:L PR[91] R[100]mm/sec CNT100;
   1:  PR[91,1] = PR[90,1] + 64.812;
   1:  PR[91,2] = PR[90,2] + -22.964;
   1:  PR[91,3] = PR[90,3] + 54.143;
   1:L PR[91] R[100]mm/sec CNT100;
   1:  PR[91,1] = PR[90,1] + 68.166;
   1:  PR[91,2] = PR[90,2] + -21.754;
   1:  PR[91,3] = PR[90,3] + 54.155;
   1:L PR[91] R[100]mm/sec CNT100;
   1:  PR[91,1] = PR[90,1] + 70.473;
   1:  PR[91,2] = PR[90,2] + -20.882;
   1:  PR[91,3] = PR[90,3] + 54.167;
   1:L PR[91] R[100]mm/sec CNT100;
   1:  PR[91,1] = PR[90,1] + 71.226;
   1:  PR[91,2] = PR[90,2] + -20.472;
   1:  PR[91,3] = PR[90,3] + 54.175;
   1:L PR[91] R[100]mm/sec CNT100;
   1:  PR[91,1] = PR[90,1] + 74.946;
   1:  PR[91,2] = PR[90,2] + -18.146;
   1:  PR[91,3] = PR[90,3] + 54.178;
   1:L PR[91] R[100]mm/sec CNT100;
   1:  PR[91,1] = PR[90,1] + 76.893;
   1:  PR[91,2] = PR[90,2] + -16.461;
   1:  PR[91,3] = PR[90,3] + 54.192;
   1:L PR[91] R[100]mm/sec CNT100;
   1:  PR[91,1] = PR[90,1] + 78.808;
   1:  PR[91,2] = PR[90,2] + -14.622;
   1:  PR[91,3] = PR[90,3] + 54.200;
   1:L PR[91] R[100]mm/sec CNT100;
   1:  PR[91,1] = PR[90,1] + 80.967;
   1:  PR[91,2] = PR[90,2] + -11.648;
   1:  PR[91,3] = PR[90,3] + 54.209;
   1:L PR[91] R[100]mm/sec CNT100;
   1:  PR[91,1] = PR[90,1] + 81.789;
   1:  PR[91,2] = PR[90,2] + -10.413;
   1:  PR[91,3] = PR[90,3] + 54.221;
   1:L PR[91] R[100]mm/sec CNT100;
   1:  PR[91,1] = PR[90,1] + 83.384;
   1:  PR[91,2] = PR[90,2] + -6.469;
   1:  PR[91,3] = PR[90,3] + 54.225;
   1:L PR[91] R[100]mm/sec CNT100;
   1:  PR[91,1] = PR[90,1] + 83.670;
   1:  PR[91,2] = PR[90,2] + -5.704;
   1:  PR[91,3] = PR[90,3] + 54.239;
   1:L PR[91] R[100]mm/sec CNT100;
   1:  PR[91,1] = PR[90,1] + 84.266;
   1:  PR[91,2] = PR[90,2] + -1.193;
   1:  PR[91,3] = PR[90,3] + 54.242;
   1:L PR[91] R[100]mm/sec CNT100;
   1:  PR[91,1] = PR[90,1] + 84.360;
   1:  PR[91,2] = PR[90,2] + -0.677;
   1:  PR[91,3] = PR[90,3] + 54.256;
   1:L PR[91] R[100]mm/sec CNT100;
   1:  PR[91,1] = PR[90,1] + 83.936;
   1:  PR[91,2] = PR[90,2] + 2.588;
   1:  PR[91,3] = PR[90,3] + 54.258;
   1:L PR[91] R[100]mm/sec CNT100;
   1:  PR[91,1] = PR[90,1] + 83.755;
   1:  PR[91,2] = PR[90,2] + 3.506;
   1:  PR[91,3] = PR[90,3] + 54.269;
   1:L PR[91] R[100]mm/sec CNT100;
   1:  PR[91,1] = PR[90,1] + 83.665;
   1:  PR[91,2] = PR[90,2] + 4.258;
   1:  PR[91,3] = PR[90,3] + 54.272;
   1:L PR[91] R[100]mm/sec CNT100;
   1:  PR[91,1] = PR[90,1] + 83.383;
   1:  PR[91,2] = PR[90,2] + 5.014;
   1:  PR[91,3] = PR[90,3] + 54.274;
   1:L PR[91] R[100]mm/sec CNT100;
   1:  PR[91,1] = PR[90,1] + 81.787;
   1:  PR[91,2] = PR[90,2] + 8.957;
   1:  PR[91,3] = PR[90,3] + 54.277;
   1:L PR[91] R[100]mm/sec CNT100;
   1:  PR[91,1] = PR[90,1] + 80.961;
   1:  PR[91,2] = PR[90,2] + 10.196;
   1:  PR[91,3] = PR[90,3] + 54.291;
   1:L PR[91] R[100]mm/sec CNT100;
   1:  PR[91,1] = PR[90,1] + 78.802;
   1:  PR[91,2] = PR[90,2] + 13.170;
   1:  PR[91,3] = PR[90,3] + 54.295;
   1:L PR[91] R[100]mm/sec CNT100;
   1:  PR[91,1] = PR[90,1] + 76.875;
   1:  PR[91,2] = PR[90,2] + 15.016;
   1:  PR[91,3] = PR[90,3] + 54.307;
   1:L PR[91] R[100]mm/sec CNT100;
   1:  PR[91,1] = PR[90,1] + 74.930;
   1:  PR[91,2] = PR[90,2] + 16.700;
   1:  PR[91,3] = PR[90,3] + 54.316;
   1:L PR[91] R[100]mm/sec CNT100;
   1:  PR[91,1] = PR[90,1] + 71.181;
   1:  PR[91,2] = PR[90,2] + 19.037;
   1:  PR[91,3] = PR[90,3] + 54.324;
   1:L PR[91] R[100]mm/sec CNT100;
   1:  PR[91,1] = PR[90,1] + 70.440;
   1:  PR[91,2] = PR[90,2] + 19.440;
   1:  PR[91,3] = PR[90,3] + 54.338;
   1:L PR[91] R[100]mm/sec CNT100;
   1:  PR[91,1] = PR[90,1] + 68.169;
   1:  PR[91,2] = PR[90,2] + 20.295;
   1:  PR[91,3] = PR[90,3] + 54.341;
   1:L PR[91] R[100]mm/sec CNT100;
   1:  PR[91,1] = PR[90,1] + 64.768;
   1:  PR[91,2] = PR[90,2] + 21.517;
   1:  PR[91,3] = PR[90,3] + 54.349;
   1:L PR[91] R[100]mm/sec CNT100;
   1:  PR[91,1] = PR[90,1] + 61.067;
   1:  PR[91,2] = PR[90,2] + 22.154;
   1:  PR[91,3] = PR[90,3] + 54.361;
   1:L PR[91] R[100]mm/sec CNT100;
   1:  PR[91,1] = PR[90,1] + 57.775;
   1:  PR[91,2] = PR[90,2] + 22.688;
   1:  PR[91,3] = PR[90,3] + 54.373;
   1:L PR[91] R[100]mm/sec CNT100;
   1:  PR[91,1] = PR[90,1] + 56.482;
   1:  PR[91,2] = PR[90,2] + 22.683;
   1:  PR[91,3] = PR[90,3] + 54.384;
   1:L PR[91] R[100]mm/sec CNT100;
   1:  PR[91,1] = PR[90,1] + 53.958;
   1:  PR[91,2] = PR[90,2] + 22.641;
   1:  PR[91,3] = PR[90,3] + 54.388;
   1:L PR[91] R[100]mm/sec CNT100;
   1:  PR[91,1] = PR[90,1] + 51.136;
   1:  PR[91,2] = PR[90,2] + 22.629;
   1:  PR[91,3] = PR[90,3] + 54.396;
   1:L PR[91] R[100]mm/sec CNT100;
   1:  PR[91,1] = PR[90,1] + 49.738;
   1:  PR[91,2] = PR[90,2] + 22.549;
   1:  PR[91,3] = PR[90,3] + 54.405;
   1:L PR[91] R[100]mm/sec CNT100;
   1:  PR[91,1] = PR[90,1] + 46.668;
   1:  PR[91,2] = PR[90,2] + 21.993;
   1:  PR[91,3] = PR[90,3] + 54.409;
   1:L PR[91] R[100]mm/sec CNT100;
   1:  PR[91,1] = PR[90,1] + 43.231;
   1:  PR[91,2] = PR[90,2] + 21.414;
   1:  PR[91,3] = PR[90,3] + 54.420;
   1:L PR[91] R[100]mm/sec CNT100;
   1:  PR[91,1] = PR[90,1] + 39.331;
   1:  PR[91,2] = PR[90,2] + 20.252;
   1:  PR[91,3] = PR[90,3] + 54.431;
   1:L PR[91] R[100]mm/sec CNT100;
   1:  PR[91,1] = PR[90,1] + 34.798;
   1:  PR[91,2] = PR[90,2] + 18.472;
   1:  PR[91,3] = PR[90,3] + 54.444;
   1:L PR[91] R[100]mm/sec CNT100;
   1:  PR[91,1] = PR[90,1] + 29.941;
   1:  PR[91,2] = PR[90,2] + 20.730;
   1:  PR[91,3] = PR[90,3] + 54.460;
   1:L PR[91] R[100]mm/sec CNT100;
   1:  PR[91,1] = PR[90,1] + 29.506;
   1:  PR[91,2] = PR[90,2] + 20.889;
   1:  PR[91,3] = PR[90,3] + 54.477;
   1:L PR[91] R[100]mm/sec CNT100;
   1:  PR[91,1] = PR[90,1] + 23.885;
   1:  PR[91,2] = PR[90,2] + 21.982;
   1:  PR[91,3] = PR[90,3] + 54.478;
   1:L PR[91] R[100]mm/sec CNT100;
   1:  PR[91,1] = PR[90,1] + 23.014;
   1:  PR[91,2] = PR[90,2] + 21.947;
   1:  PR[91,3] = PR[90,3] + 54.497;
   1:L PR[91] R[100]mm/sec CNT100;
   1:  PR[91,1] = PR[90,1] + 18.292;
   1:  PR[91,2] = PR[90,2] + 21.688;
   1:  PR[91,3] = PR[90,3] + 54.500;
   1:L PR[91] R[100]mm/sec CNT100;
   1:  PR[91,1] = PR[90,1] + 17.217;
   1:  PR[91,2] = PR[90,2] + 21.395;
   1:  PR[91,3] = PR[90,3] + 54.515;
   1:L PR[91] R[100]mm/sec CNT100;
   1:  PR[91,1] = PR[90,1] + 12.961;
   1:  PR[91,2] = PR[90,2] + 20.065;
   1:  PR[91,3] = PR[90,3] + 54.519;
   1:L PR[91] R[100]mm/sec CNT100;
   1:  PR[91,1] = PR[90,1] + 11.740;
   1:  PR[91,2] = PR[90,2] + 19.402;
   1:  PR[91,3] = PR[90,3] + 54.533;
   1:L PR[91] R[100]mm/sec CNT100;
   1:  PR[91,1] = PR[90,1] + 8.157;
   1:  PR[91,2] = PR[90,2] + 17.189;
   1:  PR[91,3] = PR[90,3] + 54.538;
   1:L PR[91] R[100]mm/sec CNT100;
   1:  PR[91,1] = PR[90,1] + 7.321;
   1:  PR[91,2] = PR[90,2] + 16.499;
   1:  PR[91,3] = PR[90,3] + 54.551;
   1:L PR[91] R[100]mm/sec CNT100;
   1:  PR[91,1] = PR[90,1] + 6.674;
   1:  PR[91,2] = PR[90,2] + 15.895;
   1:  PR[91,3] = PR[90,3] + 54.555;
   1:L PR[91] R[100]mm/sec CNT100;
   1:  PR[91,1] = PR[90,1] + 4.131;
   1:  PR[91,2] = PR[90,2] + 13.253;
   1:  PR[91,3] = PR[90,3] + 54.557;
   1:L PR[91] R[100]mm/sec CNT100;
   1:  PR[91,1] = PR[90,1] + 1.930;
   1:  PR[91,2] = PR[90,2] + 15.402;
   1:  PR[91,3] = PR[90,3] + 54.569;
   1:L PR[91] R[100]mm/sec CNT100;
   1:  PR[91,1] = PR[90,1] + 1.568;
   1:  PR[91,2] = PR[90,2] + 15.719;
   1:  PR[91,3] = PR[90,3] + 54.579;
   1:L PR[91] R[100]mm/sec CNT100;
   1:  PR[91,1] = PR[90,1] + -0.661;
   1:  PR[91,2] = PR[90,2] + 17.091;
   1:  PR[91,3] = PR[90,3] + 54.581;
   1:L PR[91] R[100]mm/sec CNT100;
   1:  PR[91,1] = PR[90,1] + -3.021;
   1:  PR[91,2] = PR[90,2] + 18.454;
   1:  PR[91,3] = PR[90,3] + 54.589;
   1:L PR[91] R[100]mm/sec CNT100;
   1:  PR[91,1] = PR[90,1] + -7.043;
   1:  PR[91,2] = PR[90,2] + 19.845;
   1:  PR[91,3] = PR[90,3] + 54.598;
   1:L PR[91] R[100]mm/sec CNT100;
   1:  PR[91,1] = PR[90,1] + -8.191;
   1:  PR[91,2] = PR[90,2] + 20.217;
   1:  PR[91,3] = PR[90,3] + 54.612;
   1:L PR[91] R[100]mm/sec CNT100;
   1:  PR[91,1] = PR[90,1] + -13.699;
   1:  PR[91,2] = PR[90,2] + 20.913;
   1:  PR[91,3] = PR[90,3] + 54.616;
   1:L PR[91] R[100]mm/sec CNT100;
   1:  PR[91,1] = PR[90,1] + -18.727;
   1:  PR[91,2] = PR[90,2] + 20.573;
   1:  PR[91,3] = PR[90,3] + 54.634;
   1:L PR[91] R[100]mm/sec CNT100;
   1:  PR[91,1] = PR[90,1] + -19.528;
   1:  PR[91,2] = PR[90,2] + 20.412;
   1:  PR[91,3] = PR[90,3] + 54.650;
   1:L PR[91] R[100]mm/sec CNT100;
   1:  PR[91,1] = PR[90,1] + -23.407;
   1:  PR[91,2] = PR[90,2] + 19.298;
   1:  PR[91,3] = PR[90,3] + 54.653;
   1:L PR[91] R[100]mm/sec CNT100;
   1:  PR[91,1] = PR[90,1] + -24.886;
   1:  PR[91,2] = PR[90,2] + 18.664;
   1:  PR[91,3] = PR[90,3] + 54.666;
   1:L PR[91] R[100]mm/sec CNT100;
   1:  PR[91,1] = PR[90,1] + -27.665;
   1:  PR[91,2] = PR[90,2] + 17.175;
   1:  PR[91,3] = PR[90,3] + 54.671;
   1:L PR[91] R[100]mm/sec CNT100;
   1:  PR[91,1] = PR[90,1] + -29.620;
   1:  PR[91,2] = PR[90,2] + 15.796;
   1:  PR[91,3] = PR[90,3] + 54.681;
   1:L PR[91] R[100]mm/sec CNT100;
   1:  PR[91,1] = PR[90,1] + -29.764;
   1:  PR[91,2] = PR[90,2] + 15.708;
   1:  PR[91,3] = PR[90,3] + 54.689;
   1:L PR[91] R[100]mm/sec CNT100;
   1:  PR[91,1] = PR[90,1] + -30.604;
   1:  PR[91,2] = PR[90,2] + 15.098;
   1:L PR[91] R[100]mm/sec CNT100;
   1:  PR[91,1] = PR[90,1] + -32.859;
   1:  PR[91,2] = PR[90,2] + 13.101;
   1:  PR[91,3] = PR[90,3] + 54.693;
   1:L PR[91] R[100]mm/sec CNT100;
   1:  PR[91,1] = PR[90,1] + -34.250;
   1:  PR[91,2] = PR[90,2] + 14.038;
   1:  PR[91,3] = PR[90,3] + 54.702;
   1:L PR[91] R[100]mm/sec CNT100;
   1:  PR[91,1] = PR[90,1] + -38.394;
   1:  PR[91,2] = PR[90,2] + 16.216;
   1:  PR[91,3] = PR[90,3] + 54.708;
   1:L PR[91] R[100]mm/sec CNT100;
   1:  PR[91,1] = PR[90,1] + -42.914;
   1:  PR[91,2] = PR[90,2] + 18.093;
   1:  PR[91,3] = PR[90,3] + 54.723;
   1:L PR[91] R[100]mm/sec CNT100;
   1:  PR[91,1] = PR[90,1] + -43.050;
   1:  PR[91,2] = PR[90,2] + 18.158;
   1:  PR[91,3] = PR[90,3] + 54.739;
   1:L PR[91] R[100]mm/sec CNT100;
   1:  PR[91,1] = PR[90,1] + -47.161;
   1:  PR[91,2] = PR[90,2] + 19.327;
   1:L PR[91] R[100]mm/sec CNT100;
   1:  PR[91,1] = PR[90,1] + -49.928;
   1:  PR[91,2] = PR[90,2] + 20.051;
   1:  PR[91,3] = PR[90,3] + 54.753;
   1:L PR[91] R[100]mm/sec CNT100;
   1:  PR[91,1] = PR[90,1] + -51.347;
   1:  PR[91,2] = PR[90,2] + 20.205;
   1:  PR[91,3] = PR[90,3] + 54.762;
   1:L PR[91] R[100]mm/sec CNT100;
   1:  PR[91,1] = PR[90,1] + -54.102;
   1:  PR[91,2] = PR[90,2] + 20.461;
   1:  PR[91,3] = PR[90,3] + 54.767;
   1:L PR[91] R[100]mm/sec CNT100;
   1:  PR[91,1] = PR[90,1] + -55.930;
   1:  PR[91,2] = PR[90,2] + 20.674;
   1:  PR[91,3] = PR[90,3] + 54.776;
   1:L PR[91] R[100]mm/sec CNT100;
   1:  PR[91,1] = PR[90,1] + -56.611;
   1:  PR[91,2] = PR[90,2] + 20.740;
   1:  PR[91,3] = PR[90,3] + 54.782;
   1:L PR[91] R[100]mm/sec CNT100;
   1:  PR[91,1] = PR[90,1] + -60.073;
   1:  PR[91,2] = PR[90,2] + 20.549;
   1:  PR[91,3] = PR[90,3] + 54.784;
   1:L PR[91] R[100]mm/sec CNT100;
   1:  PR[91] = PR[90];
   1:  PR[91,1] = PR[90,1] + -61.620;
   1:  PR[91,2] = PR[90,2] + 20.553;
   1:  PR[91,3] = PR[90,3] + 56.095;
   1:L PR[91] R[100]mm/sec CNT100;
   1:  PR[91,1] = PR[90,1] + -63.964;
   1:  PR[91,2] = PR[90,2] + 20.014;
   1:  PR[91,3] = PR[90,3] + 54.801;
   1:L PR[91] R[100]mm/sec CNT100;
   1:  PR[91,1] = PR[90,1] + -67.247;
   1:  PR[91,2] = PR[90,2] + 19.216;
   1:  PR[91,3] = PR[90,3] + 54.809;
   1:L PR[91] R[100]mm/sec CNT100;
   1:  PR[91,1] = PR[90,1] + -67.959;
   1:  PR[91,2] = PR[90,2] + 18.914;
   1:  PR[91,3] = PR[90,3] + 54.820;
   1:L PR[91] R[100]mm/sec CNT100;
   1:  PR[91,1] = PR[90,1] + -70.856;
   1:  PR[91,2] = PR[90,2] + 17.653;
   1:  PR[91,3] = PR[90,3] + 54.822;
   1:L PR[91] R[100]mm/sec CNT100;
   1:  PR[91,1] = PR[90,1] + -72.045;
   1:  PR[91,2] = PR[90,2] + 17.112;
   1:  PR[91,3] = PR[90,3] + 54.832;
   1:L PR[91] R[100]mm/sec CNT100;
   1:  PR[91,1] = PR[90,1] + -75.904;
   1:  PR[91,2] = PR[90,2] + 14.385;
   1:  PR[91,3] = PR[90,3] + 54.837;
   1:L PR[91] R[100]mm/sec CNT100;
   1:  PR[91,1] = PR[90,1] + -79.024;
   1:  PR[91,2] = PR[90,2] + 11.097;
   1:  PR[91,3] = PR[90,3] + 54.852;
   1:L PR[91] R[100]mm/sec CNT100;
   1:  PR[91,1] = PR[90,1] + -81.315;
   1:  PR[91,2] = PR[90,2] + 7.388;
   1:  PR[91,3] = PR[90,3] + 54.867;
   1:L PR[91] R[100]mm/sec CNT100;
   1:  PR[91,1] = PR[90,1] + -82.711;
   1:  PR[91,2] = PR[90,2] + 3.397;
   1:  PR[91,3] = PR[90,3] + 54.881;
   1:L PR[91] R[100]mm/sec CNT100;
   1:  PR[91,1] = PR[90,1] + -83.021;
   1:  PR[91,2] = PR[90,2] + 0.707;
   1:  PR[91,3] = PR[90,3] + 54.895;
   1:L PR[91] R[100]mm/sec CNT100;
   1:  PR[91,1] = PR[90,1] + -83.280;
   1:  PR[91,2] = PR[90,2] + -0.698;
   1:  PR[91,3] = PR[90,3] + 54.904;
   1:L PR[91] R[100]mm/sec CNT100;
   1:  PR[91,1] = PR[90,1] + -83.272;
   1:  PR[91,2] = PR[90,2] + -0.738;
   1:  PR[91,3] = PR[90,3] + 54.908;
   1:L PR[91] R[100]mm/sec CNT100;
   1:  PR[91,1] = PR[90,1] + -82.817;
   1:  PR[91,2] = PR[90,2] + -4.867;
   1:  PR[91,3] = PR[90,3] + 54.909;
   1:L PR[91] R[100]mm/sec CNT100;
   1:  PR[91,1] = PR[90,1] + -81.467;
   1:  PR[91,2] = PR[90,2] + -8.836;
   1:  PR[91,3] = PR[90,3] + 54.922;
   1:L PR[91] R[100]mm/sec CNT100;
   1:  PR[91,1] = PR[90,1] + -79.248;
   1:  PR[91,2] = PR[90,2] + -12.334;
   1:  PR[91,3] = PR[90,3] + 54.936;
   1:L PR[91] R[100]mm/sec CNT100;
   1:  PR[91,1] = PR[90,1] + -79.080;
   1:  PR[91,2] = PR[90,2] + -12.583;
   1:  PR[91,3] = PR[90,3] + 54.949;
   1:L PR[91] R[100]mm/sec CNT100;
   1:  PR[91,1] = PR[90,1] + -76.452;
   1:  PR[91,2] = PR[90,2] + -15.279;
   1:  PR[91,3] = PR[90,3] + 54.950;
   1:L PR[91] R[100]mm/sec CNT100;
   1:  PR[91,1] = PR[90,1] + -75.688;
   1:  PR[91,2] = PR[90,2] + -16.007;
   1:  PR[91,3] = PR[90,3] + 54.963;
   1:L PR[91] R[100]mm/sec CNT100;
   1:  PR[91,1] = PR[90,1] + -73.099;
   1:  PR[91,2] = PR[90,2] + -17.787;
   1:  PR[91,3] = PR[90,3] + 54.966;
   1:L PR[91] R[100]mm/sec CNT100;
   1:  PR[91,1] = PR[90,1] + -71.300;
   1:  PR[91,2] = PR[90,2] + -18.907;
   1:  PR[91,3] = PR[90,3] + 54.976;
   1:L PR[91] R[100]mm/sec CNT100;
   1:  PR[91,1] = PR[90,1] + -69.266;
   1:  PR[91,2] = PR[90,2] + -19.810;
   1:  PR[91,3] = PR[90,3] + 54.983;
   1:L PR[91] R[100]mm/sec CNT100;
   1:  PR[91,1] = PR[90,1] + -65.939;
   1:  PR[91,2] = PR[90,2] + -21.073;
   1:  PR[91,3] = PR[90,3] + 54.990;
   1:L PR[91] R[100]mm/sec CNT100;
   1:  PR[91,1] = PR[90,1] + -65.023;
   1:  PR[91,2] = PR[90,2] + -21.298;
   1:  PR[91,3] = PR[90,3] + 55.002;
   1:L PR[91] R[100]mm/sec CNT100;
   1:  PR[91,1] = PR[90,1] + -59.833;
   1:  PR[91,2] = PR[90,2] + -22.229;
   1:  PR[91,3] = PR[90,3] + 55.005;
   1:L PR[91] R[100]mm/sec CNT100;
   1:  PR[91,1] = PR[90,1] + -58.470;
   1:  PR[91,2] = PR[90,2] + -22.257;
   1:  PR[91,3] = PR[90,3] + 55.022;
   1:L PR[91] R[100]mm/sec CNT100;
   1:  PR[91,1] = PR[90,1] + -53.483;
   1:  PR[91,2] = PR[90,2] + -22.315;
   1:  PR[91,3] = PR[90,3] + 55.027;
   1:L PR[91] R[100]mm/sec CNT100;
   1:  PR[91,1] = PR[90,1] + -47.386;
   1:  PR[91,2] = PR[90,2] + -21.403;
   1:  PR[91,3] = PR[90,3] + 55.043;
   1:L PR[91] R[100]mm/sec CNT100;
   1:  PR[91,1] = PR[90,1] + -47.006;
   1:  PR[91,2] = PR[90,2] + -21.362;
   1:  PR[91,3] = PR[90,3] + 55.063;
   1:L PR[91] R[100]mm/sec CNT100;
   1:  PR[91,1] = PR[90,1] + -46.839;
   1:  PR[91,2] = PR[90,2] + -21.330;
   1:  PR[91,3] = PR[90,3] + 55.064;
   1:L PR[91] R[100]mm/sec CNT100;
   1:  PR[91,1] = PR[90,1] + -41.954;
   1:  PR[91,2] = PR[90,2] + -19.974;
   1:  PR[91,3] = PR[90,3] + 55.065;
   1:L PR[91] R[100]mm/sec CNT100;
   1:  PR[91,1] = PR[90,1] + -37.947;
   1:  PR[91,2] = PR[90,2] + -18.526;
   1:  PR[91,3] = PR[90,3] + 55.081;
   1:L PR[91] R[100]mm/sec CNT100;
   1:  PR[91,1] = PR[90,1] + -37.477;
   1:  PR[91,2] = PR[90,2] + -18.297;
   1:  PR[91,3] = PR[90,3] + 55.095;
   1:L PR[91] R[100]mm/sec CNT100;
   1:  PR[91,1] = PR[90,1] + -36.683;
   1:  PR[91,2] = PR[90,2] + -17.833;
   1:  PR[91,3] = PR[90,3] + 55.097;
   1:L PR[91] R[100]mm/sec CNT100;
   1:  PR[91,1] = PR[90,1] + -31.603;
   1:  PR[91,2] = PR[90,2] + -15.463;
   1:  PR[91,3] = PR[90,3] + 55.100;
   1:L PR[91] R[100]mm/sec CNT100;
   1:  PR[91,1] = PR[90,1] + -29.255;
   1:  PR[91,2] = PR[90,2] + -17.413;
   1:  PR[91,3] = PR[90,3] + 55.118;
   1:L PR[91] R[100]mm/sec CNT100;
   1:  PR[91,1] = PR[90,1] + -28.101;
   1:  PR[91,2] = PR[90,2] + -18.230;
   1:  PR[91,3] = PR[90,3] + 55.128;
   1:L PR[91] R[100]mm/sec CNT100;
   1:  PR[91,1] = PR[90,1] + -27.548;
   1:  PR[91,2] = PR[90,2] + -18.597;
   1:  PR[91,3] = PR[90,3] + 55.133;
   1:L PR[91] R[100]mm/sec CNT100;
   1:  PR[91,1] = PR[90,1] + -24.185;
   1:  PR[91,2] = PR[90,2] + -20.408;
   1:  PR[91,3] = PR[90,3] + 55.135;
   1:L PR[91] R[100]mm/sec CNT100;
   1:  PR[91,1] = PR[90,1] + -23.220;
   1:  PR[91,2] = PR[90,2] + -20.822;
   1:  PR[91,3] = PR[90,3] + 55.148;
   1:L PR[91] R[100]mm/sec CNT100;
   1:  PR[91,1] = PR[90,1] + -18.736;
   1:  PR[91,2] = PR[90,2] + -22.118;
   1:  PR[91,3] = PR[90,3] + 55.151;
   1:L PR[91] R[100]mm/sec CNT100;
   1:  PR[91,1] = PR[90,1] + -18.518;
   1:  PR[91,2] = PR[90,2] + -22.162;
   1:  PR[91,3] = PR[90,3] + 55.166;
   1:L PR[91] R[100]mm/sec CNT100;
   1:  PR[91,1] = PR[90,1] + -16.191;
   1:  PR[91,2] = PR[90,2] + -22.325;
   1:  PR[91,3] = PR[90,3] + 55.167;
   1:L PR[91] R[100]mm/sec CNT100;
   1:  PR[91,1] = PR[90,1] + -13.108;
   1:  PR[91,2] = PR[90,2] + -22.571;
   1:  PR[91,3] = PR[90,3] + 55.175;
   1:L PR[91] R[100]mm/sec CNT100;
   1:  PR[91,1] = PR[90,1] + -8.844;
   1:  PR[91,2] = PR[90,2] + -22.035;
   1:  PR[91,3] = PR[90,3] + 55.185;
   1:L PR[91] R[100]mm/sec CNT100;
   1:  PR[91,1] = PR[90,1] + -7.533;
   1:  PR[91,2] = PR[90,2] + -21.887;
   1:  PR[91,3] = PR[90,3] + 55.199;
   1:L PR[91] R[100]mm/sec CNT100;
   1:  PR[91,1] = PR[90,1] + -5.457;
   1:  PR[91,2] = PR[90,2] + -21.215;
   1:  PR[91,3] = PR[90,3] + 55.203;
   1:L PR[91] R[100]mm/sec CNT100;
   1:  PR[91,1] = PR[90,1] + -2.356;
   1:  PR[91,2] = PR[90,2] + -20.147;
   1:  PR[91,3] = PR[90,3] + 55.210;
   1:L PR[91] R[100]mm/sec CNT100;
   1:  PR[91,1] = PR[90,1] + 0.847;
   1:  PR[91,2] = PR[90,2] + -18.306;
   1:  PR[91,3] = PR[90,3] + 55.221;
   1:L PR[91] R[100]mm/sec CNT100;
   1:  PR[91,1] = PR[90,1] + 2.228;
   1:  PR[91,2] = PR[90,2] + -17.458;
   1:  PR[91,3] = PR[90,3] + 55.233;
   1:L PR[91] R[100]mm/sec CNT100;
   1:  PR[91,1] = PR[90,1] + 4.365;
   1:  PR[91,2] = PR[90,2] + -15.477;
   1:  PR[91,3] = PR[90,3] + 55.238;
   1:L PR[91] R[100]mm/sec CNT100;
   1:  PR[91,1] = PR[90,1] + 6.936;
   1:  PR[91,2] = PR[90,2] + -18.027;
   1:  PR[91,3] = PR[90,3] + 55.248;
   1:L PR[91] R[100]mm/sec CNT100;
   1:  PR[91,1] = PR[90,1] + 7.370;
   1:  PR[91,2] = PR[90,2] + -18.408;
   1:  PR[91,3] = PR[90,3] + 55.259;
   1:L PR[91] R[100]mm/sec CNT100;
   1:  PR[91,1] = PR[90,1] + 7.993;
   1:  PR[91,2] = PR[90,2] + -18.897;
   1:  PR[91,3] = PR[90,3] + 55.261;
   1:L PR[91] R[100]mm/sec CNT100;
   1:  PR[91,1] = PR[90,1] + 11.098;
   1:  PR[91,2] = PR[90,2] + -20.817;
   1:  PR[91,3] = PR[90,3] + 55.264;
   1:L PR[91] R[100]mm/sec CNT100;
   1:  PR[91,1] = PR[90,1] + 12.831;
   1:  PR[91,2] = PR[90,2] + -21.756;
   1:  PR[91,3] = PR[90,3] + 55.276;
   1:L PR[91] R[100]mm/sec CNT100;
   1:  PR[91,1] = PR[90,1] + 16.535;
   1:  PR[91,2] = PR[90,2] + -22.915;
   1:  PR[91,3] = PR[90,3] + 55.282;
   1:L PR[91] R[100]mm/sec CNT100;
   1:  PR[91,1] = PR[90,1] + 18.166;
   1:  PR[91,2] = PR[90,2] + -23.360;
   1:  PR[91,3] = PR[90,3] + 55.295;
   1:L PR[91] R[100]mm/sec CNT100;
   1:  PR[91,1] = PR[90,1] + 22.316;
   1:  PR[91,2] = PR[90,2] + -23.589;
   1:  PR[91,3] = PR[90,3] + 55.300;
   1:L PR[91] R[100]mm/sec CNT100;
   1:  PR[91,1] = PR[90,1] + 23.758;
   1:  PR[91,2] = PR[90,2] + -23.646;
   1:  PR[91,3] = PR[90,3] + 55.314;
   1:L PR[91] R[100]mm/sec CNT100;
   1:  PR[91,1] = PR[90,1] + 29.429;
   1:  PR[91,2] = PR[90,2] + -22.546;
   1:  PR[91,3] = PR[90,3] + 55.319;
   1:L PR[91] R[100]mm/sec CNT100;
   1:  PR[91,1] = PR[90,1] + 29.654;
   1:  PR[91,2] = PR[90,2] + -22.473;
   1:  PR[91,3] = PR[90,3] + 55.337;
   1:L PR[91] R[100]mm/sec CNT100;
   1:  PR[91,1] = PR[90,1] + 30.242;
   1:  PR[91,2] = PR[90,2] + -22.245;
   1:  PR[91,3] = PR[90,3] + 55.338;
   1:L PR[91] R[100]mm/sec CNT100;
   1:  PR[91,1] = PR[90,1] + 34.121;
   1:  PR[91,2] = PR[90,2] + -20.442;
   1:  PR[91,3] = PR[90,3] + 55.340;
   1:L PR[91] R[100]mm/sec CNT100;
   1:  PR[91,1] = PR[90,1] + 38.678;
   1:  PR[91,2] = PR[90,2] + -22.231;
   1:  PR[91,3] = PR[90,3] + 55.354;
   1:L PR[91] R[100]mm/sec CNT100;
   1:  PR[91,1] = PR[90,1] + 39.878;
   1:  PR[91,2] = PR[90,2] + -22.587;
   1:  PR[91,3] = PR[90,3] + 55.370;
   1:L PR[91] R[100]mm/sec CNT100;
   1:  PR[91,1] = PR[90,1] + 42.532;
   1:  PR[91,2] = PR[90,2] + -23.258;
   1:  PR[91,3] = PR[90,3] + 55.374;
   1:L PR[91] R[100]mm/sec CNT100;
   1:  PR[91,1] = PR[90,1] + 44.182;
   1:  PR[91,2] = PR[90,2] + -23.526;
   1:  PR[91,3] = PR[90,3] + 55.383;
   1:L PR[91] R[100]mm/sec CNT100;
   1:  PR[91,1] = PR[90,1] + 48.113;
   1:  PR[91,2] = PR[90,2] + -24.212;
   1:  PR[91,3] = PR[90,3] + 55.389;
   1:L PR[91] R[100]mm/sec CNT100;
   1:  PR[91,1] = PR[90,1] + 50.621;
   1:  PR[91,2] = PR[90,2] + -24.356;
   1:  PR[91,3] = PR[90,3] + 55.402;
   1:L PR[91] R[100]mm/sec CNT100;
   1:  PR[91,1] = PR[90,1] + 56.624;
   1:  PR[91,2] = PR[90,2] + -24.396;
   1:  PR[91,3] = PR[90,3] + 55.410;
   1:L PR[91] R[100]mm/sec CNT100;
   1:  PR[91,1] = PR[90,1] + 60.917;
   1:  PR[91,2] = PR[90,2] + -23.705;
   1:  PR[91,3] = PR[90,3] + 55.429;
   1:L PR[91] R[100]mm/sec CNT100;
   1:  PR[91,1] = PR[90,1] + 63.769;
   1:  PR[91,2] = PR[90,2] + -23.207;
   1:  PR[91,3] = PR[90,3] + 55.444;
   1:L PR[91] R[100]mm/sec CNT100;
   1:  PR[91,1] = PR[90,1] + 65.463;
   1:  PR[91,2] = PR[90,2] + -22.611;
   1:  PR[91,3] = PR[90,3] + 55.453;
   1:L PR[91] R[100]mm/sec CNT100;
   1:  PR[91,1] = PR[90,1] + 70.005;
   1:  PR[91,2] = PR[90,2] + -20.956;
   1:  PR[91,3] = PR[90,3] + 55.459;
   1:L PR[91] R[100]mm/sec CNT100;
   1:  PR[91,1] = PR[90,1] + 74.473;
   1:  PR[91,2] = PR[90,2] + -18.165;
   1:  PR[91,3] = PR[90,3] + 55.475;
   1:L PR[91] R[100]mm/sec CNT100;
   1:  PR[91,1] = PR[90,1] + 75.727;
   1:  PR[91,2] = PR[90,2] + -17.080;
   1:  PR[91,3] = PR[90,3] + 55.492;
   1:L PR[91] R[100]mm/sec CNT100;
   1:  PR[91,1] = PR[90,1] + 78.290;
   1:  PR[91,2] = PR[90,2] + -14.619;
   1:  PR[91,3] = PR[90,3] + 55.497;
   1:L PR[91] R[100]mm/sec CNT100;
   1:  PR[91,1] = PR[90,1] + 79.961;
   1:  PR[91,2] = PR[90,2] + -12.317;
   1:  PR[91,3] = PR[90,3] + 55.509;
   1:L PR[91] R[100]mm/sec CNT100;
   1:  PR[91,1] = PR[90,1] + 81.235;
   1:  PR[91,2] = PR[90,2] + -10.403;
   1:  PR[91,3] = PR[90,3] + 55.518;
   1:L PR[91] R[100]mm/sec CNT100;
   1:  PR[91,1] = PR[90,1] + 82.548;
   1:  PR[91,2] = PR[90,2] + -7.159;
   1:  PR[91,3] = PR[90,3] + 55.526;
   1:L PR[91] R[100]mm/sec CNT100;
   1:  PR[91,1] = PR[90,1] + 83.094;
   1:  PR[91,2] = PR[90,2] + -5.697;
   1:  PR[91,3] = PR[90,3] + 55.537;
   1:L PR[91] R[100]mm/sec CNT100;
   1:  PR[91,1] = PR[90,1] + 83.597;
   1:  PR[91,2] = PR[90,2] + -1.884;
   1:  PR[91,3] = PR[90,3] + 55.542;
   1:L PR[91] R[100]mm/sec CNT100;
   1:  PR[91,1] = PR[90,1] + 83.819;
   1:  PR[91,2] = PR[90,2] + -0.677;
   1:  PR[91,3] = PR[90,3] + 55.555;
   1:L PR[91] R[100]mm/sec CNT100;
   1:  PR[91,1] = PR[90,1] + 83.560;
   1:  PR[91,2] = PR[90,2] + 1.315;
   1:  PR[91,3] = PR[90,3] + 55.559;
   1:L PR[91] R[100]mm/sec CNT100;
   1:  PR[91,1] = PR[90,1] + 83.254;
   1:  PR[91,2] = PR[90,2] + 2.863;
   1:  PR[91,3] = PR[90,3] + 55.565;
   1:L PR[91] R[100]mm/sec CNT100;
   1:  PR[91,1] = PR[90,1] + 83.089;
   1:  PR[91,2] = PR[90,2] + 4.252;
   1:  PR[91,3] = PR[90,3] + 55.570;
   1:L PR[91] R[100]mm/sec CNT100;
   1:  PR[91,1] = PR[90,1] + 82.545;
   1:  PR[91,2] = PR[90,2] + 5.706;
   1:  PR[91,3] = PR[90,3] + 55.575;
   1:L PR[91] R[100]mm/sec CNT100;
   1:  PR[91,1] = PR[90,1] + 81.233;
   1:  PR[91,2] = PR[90,2] + 8.950;
   1:  PR[91,3] = PR[90,3] + 55.580;
   1:L PR[91] R[100]mm/sec CNT100;
   1:  PR[91,1] = PR[90,1] + 79.952;
   1:  PR[91,2] = PR[90,2] + 10.869;
   1:  PR[91,3] = PR[90,3] + 55.591;
   1:L PR[91] R[100]mm/sec CNT100;
   1:  PR[91,1] = PR[90,1] + 78.281;
   1:  PR[91,2] = PR[90,2] + 13.171;
   1:  PR[91,3] = PR[90,3] + 55.599;
   1:L PR[91] R[100]mm/sec CNT100;
   1:  PR[91,1] = PR[90,1] + 75.703;
   1:  PR[91,2] = PR[90,2] + 15.640;
   1:  PR[91,3] = PR[90,3] + 55.608;
   1:L PR[91] R[100]mm/sec CNT100;
   1:  PR[91,1] = PR[90,1] + 74.453;
   1:  PR[91,2] = PR[90,2] + 16.722;
   1:  PR[91,3] = PR[90,3] + 55.620;
   1:L PR[91] R[100]mm/sec CNT100;
   1:  PR[91,1] = PR[90,1] + 69.968;
   1:  PR[91,2] = PR[90,2] + 19.517;
   1:  PR[91,3] = PR[90,3] + 55.625;
   1:L PR[91] R[100]mm/sec CNT100;
   1:  PR[91,1] = PR[90,1] + 65.432;
   1:  PR[91,2] = PR[90,2] + 21.158;
   1:  PR[91,3] = PR[90,3] + 55.643;
   1:L PR[91] R[100]mm/sec CNT100;
   1:  PR[91,1] = PR[90,1] + 63.740;
   1:  PR[91,2] = PR[90,2] + 21.756;
   1:  PR[91,3] = PR[90,3] + 55.658;
   1:L PR[91] R[100]mm/sec CNT100;
   1:  PR[91,1] = PR[90,1] + 60.904;
   1:  PR[91,2] = PR[90,2] + 22.244;
   1:  PR[91,3] = PR[90,3] + 55.664;
   1:L PR[91] R[100]mm/sec CNT100;
   1:  PR[91,1] = PR[90,1] + 56.645;
   1:  PR[91,2] = PR[90,2] + 22.935;
   1:  PR[91,3] = PR[90,3] + 55.674;
   1:L PR[91] R[100]mm/sec CNT100;
   1:  PR[91,1] = PR[90,1] + 50.639;
   1:  PR[91,2] = PR[90,2] + 22.900;
   1:  PR[91,3] = PR[90,3] + 55.688;
   1:L PR[91] R[100]mm/sec CNT100;
   1:  PR[91,1] = PR[90,1] + 48.137;
   1:  PR[91,2] = PR[90,2] + 22.756;
   1:  PR[91,3] = PR[90,3] + 55.707;
   1:L PR[91] R[100]mm/sec CNT100;
   1:  PR[91,1] = PR[90,1] + 46.362;
   1:  PR[91,2] = PR[90,2] + 22.434;
   1:  PR[91,3] = PR[90,3] + 55.715;
   1:L PR[91] R[100]mm/sec CNT100;
   1:  PR[91,1] = PR[90,1] + 42.536;
   1:  PR[91,2] = PR[90,2] + 21.800;
   1:  PR[91,3] = PR[90,3] + 55.721;
   1:L PR[91] R[100]mm/sec CNT100;
   1:  PR[91,1] = PR[90,1] + 39.878;
   1:  PR[91,2] = PR[90,2] + 21.128;
   1:  PR[91,3] = PR[90,3] + 55.734;
   1:L PR[91] R[100]mm/sec CNT100;
   1:  PR[91,1] = PR[90,1] + 38.678;
   1:  PR[91,2] = PR[90,2] + 20.772;
   1:  PR[91,3] = PR[90,3] + 55.743;
   1:L PR[91] R[100]mm/sec CNT100;
   1:  PR[91,1] = PR[90,1] + 34.121;
   1:  PR[91,2] = PR[90,2] + 18.984;
   1:  PR[91,3] = PR[90,3] + 55.747;
   1:L PR[91] R[100]mm/sec CNT100;
   1:  PR[91,1] = PR[90,1] + 30.243;
   1:  PR[91,2] = PR[90,2] + 20.786;
   1:  PR[91,3] = PR[90,3] + 55.763;
   1:L PR[91] R[100]mm/sec CNT100;
   1:  PR[91,1] = PR[90,1] + 29.656;
   1:  PR[91,2] = PR[90,2] + 21.013;
   1:  PR[91,3] = PR[90,3] + 55.777;
   1:L PR[91] R[100]mm/sec CNT100;
   1:  PR[91,1] = PR[90,1] + 29.429;
   1:  PR[91,2] = PR[90,2] + 21.088;
   1:  PR[91,3] = PR[90,3] + 55.779;
   1:L PR[91] R[100]mm/sec CNT100;
   1:  PR[91,1] = PR[90,1] + 25.050;
   1:  PR[91,2] = PR[90,2] + 21.947;
   1:  PR[91,3] = PR[90,3] + 55.780;
   1:L PR[91] R[100]mm/sec CNT100;
   1:  PR[91,1] = PR[90,1] + 23.769;
   1:  PR[91,2] = PR[90,2] + 22.187;
   1:  PR[91,3] = PR[90,3] + 55.794;
   1:L PR[91] R[100]mm/sec CNT100;
   1:  PR[91,1] = PR[90,1] + 22.319;
   1:  PR[91,2] = PR[90,2] + 22.129;
   1:  PR[91,3] = PR[90,3] + 55.799;
   1:L PR[91] R[100]mm/sec CNT100;
   1:  PR[91,1] = PR[90,1] + 18.172;
   1:  PR[91,2] = PR[90,2] + 21.902;
   1:  PR[91,3] = PR[90,3] + 55.803;
   1:L PR[91] R[100]mm/sec CNT100;
   1:  PR[91,1] = PR[90,1] + 16.540;
   1:  PR[91,2] = PR[90,2] + 21.457;
   1:  PR[91,3] = PR[90,3] + 55.817;
   1:L PR[91] R[100]mm/sec CNT100;
   1:  PR[91,1] = PR[90,1] + 12.837;
   1:  PR[91,2] = PR[90,2] + 20.300;
   1:  PR[91,3] = PR[90,3] + 55.822;
   1:L PR[91] R[100]mm/sec CNT100;
   1:  PR[91,1] = PR[90,1] + 11.093;
   1:  PR[91,2] = PR[90,2] + 19.354;
   1:  PR[91,3] = PR[90,3] + 55.835;
   1:L PR[91] R[100]mm/sec CNT100;
   1:  PR[91,1] = PR[90,1] + 8.016;
   1:  PR[91,2] = PR[90,2] + 17.453;
   1:  PR[91,3] = PR[90,3] + 55.841;
   1:L PR[91] R[100]mm/sec CNT100;
   1:  PR[91,1] = PR[90,1] + 6.862;
   1:  PR[91,2] = PR[90,2] + 16.500;
   1:  PR[91,3] = PR[90,3] + 55.853;
   1:L PR[91] R[100]mm/sec CNT100;
   1:  PR[91,1] = PR[90,1] + 5.980;
   1:  PR[91,2] = PR[90,2] + 15.676;
   1:  PR[91,3] = PR[90,3] + 55.858;
   1:L PR[91] R[100]mm/sec CNT100;
   1:  PR[91,1] = PR[90,1] + 4.353;
   1:  PR[91,2] = PR[90,2] + 13.986;
   1:  PR[91,3] = PR[90,3] + 55.862;
   1:L PR[91] R[100]mm/sec CNT100;
   1:  PR[91,1] = PR[90,1] + 2.769;
   1:  PR[91,2] = PR[90,2] + 15.532;
   1:  PR[91,3] = PR[90,3] + 55.870;
   1:L PR[91] R[100]mm/sec CNT100;
   1:  PR[91,1] = PR[90,1] + 2.279;
   1:  PR[91,2] = PR[90,2] + 15.962;
   1:  PR[91,3] = PR[90,3] + 55.877;
   1:L PR[91] R[100]mm/sec CNT100;
   1:  PR[91,1] = PR[90,1] + 0.916;
   1:  PR[91,2] = PR[90,2] + 16.801;
   1:  PR[91,3] = PR[90,3] + 55.879;
   1:L PR[91] R[100]mm/sec CNT100;
   1:  PR[91,1] = PR[90,1] + -2.335;
   1:  PR[91,2] = PR[90,2] + 18.678;
   1:  PR[91,3] = PR[90,3] + 55.884;
   1:L PR[91] R[100]mm/sec CNT100;
   1:  PR[91,1] = PR[90,1] + -5.422;
   1:  PR[91,2] = PR[90,2] + 19.746;
   1:  PR[91,3] = PR[90,3] + 55.897;
   1:L PR[91] R[100]mm/sec CNT100;
   1:  PR[91,1] = PR[90,1] + -7.514;
   1:  PR[91,2] = PR[90,2] + 20.425;
   1:  PR[91,3] = PR[90,3] + 55.907;
   1:L PR[91] R[100]mm/sec CNT100;
   1:  PR[91,1] = PR[90,1] + -13.070;
   1:  PR[91,2] = PR[90,2] + 21.112;
   1:  PR[91,3] = PR[90,3] + 55.914;
   1:L PR[91] R[100]mm/sec CNT100;
   1:  PR[91,1] = PR[90,1] + -16.194;
   1:  PR[91,2] = PR[90,2] + 20.867;
   1:  PR[91,3] = PR[90,3] + 55.933;
   1:L PR[91] R[100]mm/sec CNT100;
   1:  PR[91,1] = PR[90,1] + -18.484;
   1:  PR[91,2] = PR[90,2] + 20.709;
   1:  PR[91,3] = PR[90,3] + 55.943;
   1:L PR[91] R[100]mm/sec CNT100;
   1:  PR[91,1] = PR[90,1] + -18.696;
   1:  PR[91,2] = PR[90,2] + 20.666;
   1:  PR[91,3] = PR[90,3] + 55.950;
   1:L PR[91] R[100]mm/sec CNT100;
   1:  PR[91,1] = PR[90,1] + -23.191;
   1:  PR[91,2] = PR[90,2] + 19.376;
   1:  PR[91,3] = PR[90,3] + 55.951;
   1:L PR[91] R[100]mm/sec CNT100;
   1:  PR[91,1] = PR[90,1] + -24.152;
   1:  PR[91,2] = PR[90,2] + 18.964;
   1:  PR[91,3] = PR[90,3] + 55.966;
   1:L PR[91] R[100]mm/sec CNT100;
   1:  PR[91,1] = PR[90,1] + -27.459;
   1:  PR[91,2] = PR[90,2] + 17.191;
   1:  PR[91,3] = PR[90,3] + 55.970;
   1:L PR[91] R[100]mm/sec CNT100;
   1:  PR[91,1] = PR[90,1] + -28.982;
   1:  PR[91,2] = PR[90,2] + 16.117;
   1:  PR[91,3] = PR[90,3] + 55.982;
   1:L PR[91] R[100]mm/sec CNT100;
   1:  PR[91,1] = PR[90,1] + -29.160;
   1:  PR[91,2] = PR[90,2] + 16.009;
   1:  PR[91,3] = PR[90,3] + 55.988;
   1:L PR[91] R[100]mm/sec CNT100;
   1:  PR[91,1] = PR[90,1] + -30.212;
   1:  PR[91,2] = PR[90,2] + 15.245;
   1:  PR[91,3] = PR[90,3] + 55.989;
   1:L PR[91] R[100]mm/sec CNT100;
   1:  PR[91,1] = PR[90,1] + -31.561;
   1:  PR[91,2] = PR[90,2] + 14.061;
   1:  PR[91,3] = PR[90,3] + 55.993;
   1:L PR[91] R[100]mm/sec CNT100;
   1:  PR[91,1] = PR[90,1] + -34.657;
   1:  PR[91,2] = PR[90,2] + 15.314;
   1:  PR[91,3] = PR[90,3] + 55.999;
   1:L PR[91] R[100]mm/sec CNT100;
   1:  PR[91,1] = PR[90,1] + -37.621;
   1:  PR[91,2] = PR[90,2] + 16.871;
   1:  PR[91,3] = PR[90,3] + 56.010;
   1:L PR[91] R[100]mm/sec CNT100;
   1:  PR[91,1] = PR[90,1] + -40.482;
   1:  PR[91,2] = PR[90,2] + 18.059;
   1:  PR[91,3] = PR[90,3] + 56.021;
   1:L PR[91] R[100]mm/sec CNT100;
   1:  PR[91,1] = PR[90,1] + -42.128;
   1:  PR[91,2] = PR[90,2] + 18.560;
   1:  PR[91,3] = PR[90,3] + 56.031;
   1:L PR[91] R[100]mm/sec CNT100;
   1:  PR[91,1] = PR[90,1] + -43.916;
   1:  PR[91,2] = PR[90,2] + 18.973;
   1:  PR[91,3] = PR[90,3] + 56.036;
   1:L PR[91] R[100]mm/sec CNT100;
   1:  PR[91,1] = PR[90,1] + -46.788;
   1:  PR[91,2] = PR[90,2] + 19.789;
   1:  PR[91,3] = PR[90,3] + 56.042;
   1:L PR[91] R[100]mm/sec CNT100;
   1:  PR[91,1] = PR[90,1] + -48.459;
   1:  PR[91,2] = PR[90,2] + 20.226;
   1:  PR[91,3] = PR[90,3] + 56.052;
   1:L PR[91] R[100]mm/sec CNT100;
   1:  PR[91,1] = PR[90,1] + -51.020;
   1:  PR[91,2] = PR[90,2] + 20.505;
   1:  PR[91,3] = PR[90,3] + 56.058;
   1:L PR[91] R[100]mm/sec CNT100;
   1:  PR[91,1] = PR[90,1] + -55.495;
   1:  PR[91,2] = PR[90,2] + 20.921;
   1:  PR[91,3] = PR[90,3] + 56.066;
   1:L PR[91] R[100]mm/sec CNT100;
   1:  PR[91,1] = PR[90,1] + -59.861;
   1:  PR[91,2] = PR[90,2] + 20.678;
   1:  PR[91,3] = PR[90,3] + 56.081;
   1:L PR[91] R[100]mm/sec CNT100;
   1:  PR[91] = PR[90];
   1:  PR[91,1] = PR[90,1] + -60.598;
   1:  PR[91,2] = PR[90,2] + 20.741;
   1:  PR[91,3] = PR[90,3] + 57.395;
   1:L PR[91] R[100]mm/sec CNT100;
   1:  PR[91,1] = PR[90,1] + -63.743;
   1:  PR[91,2] = PR[90,2] + 20.018;
   1:  PR[91,3] = PR[90,3] + 56.098;
   1:L PR[91] R[100]mm/sec CNT100;
   1:  PR[91,1] = PR[90,1] + -66.296;
   1:  PR[91,2] = PR[90,2] + 19.396;
   1:  PR[91,3] = PR[90,3] + 56.109;
   1:L PR[91] R[100]mm/sec CNT100;
   1:  PR[91,1] = PR[90,1] + -67.707;
   1:  PR[91,2] = PR[90,2] + 18.799;
   1:  PR[91,3] = PR[90,3] + 56.117;
   1:L PR[91] R[100]mm/sec CNT100;
   1:  PR[91,1] = PR[90,1] + -71.319;
   1:  PR[91,2] = PR[90,2] + 17.227;
   1:  PR[91,3] = PR[90,3] + 56.122;
   1:L PR[91] R[100]mm/sec CNT100;
   1:  PR[91,1] = PR[90,1] + -72.625;
   1:  PR[91,2] = PR[90,2] + 16.353;
   1:  PR[91,3] = PR[90,3] + 56.135;
   1:L PR[91] R[100]mm/sec CNT100;
   1:  PR[91,1] = PR[90,1] + -75.283;
   1:  PR[91,2] = PR[90,2] + 14.472;
   1:  PR[91,3] = PR[90,3] + 56.141;
   1:L PR[91] R[100]mm/sec CNT100;
   1:  PR[91,1] = PR[90,1] + -78.417;
   1:  PR[91,2] = PR[90,2] + 11.164;
   1:  PR[91,3] = PR[90,3] + 56.151;
   1:L PR[91] R[100]mm/sec CNT100;
   1:  PR[91,1] = PR[90,1] + -80.717;
   1:  PR[91,2] = PR[90,2] + 7.433;
   1:  PR[91,3] = PR[90,3] + 56.166;
   1:L PR[91] R[100]mm/sec CNT100;
   1:  PR[91,1] = PR[90,1] + -82.119;
   1:  PR[91,2] = PR[90,2] + 3.420;
   1:  PR[91,3] = PR[90,3] + 56.181;
   1:L PR[91] R[100]mm/sec CNT100;
   1:  PR[91,1] = PR[90,1] + -82.361;
   1:  PR[91,2] = PR[90,2] + 1.315;
   1:  PR[91,3] = PR[90,3] + 56.195;
   1:L PR[91] R[100]mm/sec CNT100;
   1:  PR[91,1] = PR[90,1] + -82.734;
   1:  PR[91,2] = PR[90,2] + -0.703;
   1:  PR[91,3] = PR[90,3] + 56.202;
   1:L PR[91] R[100]mm/sec CNT100;
   1:  PR[91,1] = PR[90,1] + -82.742;
   1:  PR[91,2] = PR[90,2] + -0.761;
   1:  PR[91,3] = PR[90,3] + 56.209;
   1:L PR[91] R[100]mm/sec CNT100;
   1:  PR[91,1] = PR[90,1] + -82.483;
   1:  PR[91,2] = PR[90,2] + -3.036;
   1:L PR[91] R[100]mm/sec CNT100;
   1:  PR[91,1] = PR[90,1] + -82.302;
   1:  PR[91,2] = PR[90,2] + -4.479;
   1:  PR[91,3] = PR[90,3] + 56.216;
   1:L PR[91] R[100]mm/sec CNT100;
   1:  PR[91,1] = PR[90,1] + -82.250;
   1:  PR[91,2] = PR[90,2] + -4.726;
   1:  PR[91,3] = PR[90,3] + 56.221;
   1:L PR[91] R[100]mm/sec CNT100;
   1:  PR[91,1] = PR[90,1] + -82.232;
   1:  PR[91,2] = PR[90,2] + -4.874;
   1:  PR[91,3] = PR[90,3] + 56.222;
   1:L PR[91] R[100]mm/sec CNT100;
   1:  PR[91,1] = PR[90,1] + -80.766;
   1:  PR[91,2] = PR[90,2] + -8.928;
   1:L PR[91] R[100]mm/sec CNT100;
   1:  PR[91,1] = PR[90,1] + -78.820;
   1:  PR[91,2] = PR[90,2] + -11.996;
   1:  PR[91,3] = PR[90,3] + 56.237;
   1:L PR[91] R[100]mm/sec CNT100;
   1:  PR[91,1] = PR[90,1] + -78.320;
   1:  PR[91,2] = PR[90,2] + -12.740;
   1:  PR[91,3] = PR[90,3] + 56.249;
   1:L PR[91] R[100]mm/sec CNT100;
   1:  PR[91,1] = PR[90,1] + -76.080;
   1:  PR[91,2] = PR[90,2] + -15.037;
   1:  PR[91,3] = PR[90,3] + 56.252;
   1:L PR[91] R[100]mm/sec CNT100;
   1:  PR[91,1] = PR[90,1] + -74.857;
   1:  PR[91,2] = PR[90,2] + -16.203;
   1:  PR[91,3] = PR[90,3] + 56.262;
   1:L PR[91] R[100]mm/sec CNT100;
   1:  PR[91,1] = PR[90,1] + -72.762;
   1:  PR[91,2] = PR[90,2] + -17.643;
   1:  PR[91,3] = PR[90,3] + 56.268;
   1:L PR[91] R[100]mm/sec CNT100;
   1:  PR[91,1] = PR[90,1] + -70.376;
   1:  PR[91,2] = PR[90,2] + -19.129;
   1:  PR[91,3] = PR[90,3] + 56.276;
   1:L PR[91] R[100]mm/sec CNT100;
   1:  PR[91,1] = PR[90,1] + -68.942;
   1:  PR[91,2] = PR[90,2] + -19.765;
   1:  PR[91,3] = PR[90,3] + 56.285;
   1:L PR[91] R[100]mm/sec CNT100;
   1:  PR[91,1] = PR[90,1] + -64.899;
   1:  PR[91,2] = PR[90,2] + -21.301;
   1:  PR[91,3] = PR[90,3] + 56.291;
   1:L PR[91] R[100]mm/sec CNT100;
   1:  PR[91,1] = PR[90,1] + -64.690;
   1:  PR[91,2] = PR[90,2] + -21.352;
   1:  PR[91,3] = PR[90,3] + 56.305;
   1:L PR[91] R[100]mm/sec CNT100;
   1:  PR[91,1] = PR[90,1] + -58.819;
   1:  PR[91,2] = PR[90,2] + -22.413;
   1:  PR[91,3] = PR[90,3] + 56.306;
   1:L PR[91] R[100]mm/sec CNT100;
   1:  PR[91,1] = PR[90,1] + -55.344;
   1:  PR[91,2] = PR[90,2] + -22.485;
   1:  PR[91,3] = PR[90,3] + 56.325;
   1:L PR[91] R[100]mm/sec CNT100;
   1:  PR[91,1] = PR[90,1] + -52.420;
   1:  PR[91,2] = PR[90,2] + -22.519;
   1:  PR[91,3] = PR[90,3] + 56.337;
   1:L PR[91] R[100]mm/sec CNT100;
   1:  PR[91,1] = PR[90,1] + -48.811;
   1:  PR[91,2] = PR[90,2] + -21.979;
   1:  PR[91,3] = PR[90,3] + 56.346;
   1:L PR[91] R[100]mm/sec CNT100;
   1:  PR[91,1] = PR[90,1] + -46.253;
   1:  PR[91,2] = PR[90,2] + -21.699;
   1:  PR[91,3] = PR[90,3] + 56.358;
   1:L PR[91] R[100]mm/sec CNT100;
   1:  PR[91,1] = PR[90,1] + -44.402;
   1:  PR[91,2] = PR[90,2] + -21.344;
   1:  PR[91,3] = PR[90,3] + 56.367;
   1:L PR[91] R[100]mm/sec CNT100;
   1:  PR[91,1] = PR[90,1] + -41.197;
   1:  PR[91,2] = PR[90,2] + -20.455;
   1:  PR[91,3] = PR[90,3] + 56.373;
   1:L PR[91] R[100]mm/sec CNT100;
   1:  PR[91,1] = PR[90,1] + -37.462;
   1:  PR[91,2] = PR[90,2] + -19.105;
   1:  PR[91,3] = PR[90,3] + 56.384;
   1:L PR[91] R[100]mm/sec CNT100;
   1:  PR[91,1] = PR[90,1] + -36.263;
   1:  PR[91,2] = PR[90,2] + -18.766;
   1:  PR[91,3] = PR[90,3] + 56.397;
   1:L PR[91] R[100]mm/sec CNT100;
   1:  PR[91,1] = PR[90,1] + -35.098;
   1:  PR[91,2] = PR[90,2] + -18.345;
   1:  PR[91,3] = PR[90,3] + 56.401;
   1:L PR[91] R[100]mm/sec CNT100;
   1:  PR[91,1] = PR[90,1] + -30.488;
   1:  PR[91,2] = PR[90,2] + -16.194;
   1:  PR[91,3] = PR[90,3] + 56.405;
   1:L PR[91] R[100]mm/sec CNT100;
   1:  PR[91,1] = PR[90,1] + -28.685;
   1:  PR[91,2] = PR[90,2] + -17.692;
   1:  PR[91,3] = PR[90,3] + 56.422;
   1:L PR[91] R[100]mm/sec CNT100;
   1:  PR[91,1] = PR[90,1] + -28.003;
   1:  PR[91,2] = PR[90,2] + -18.175;
   1:  PR[91,3] = PR[90,3] + 56.430;
   1:L PR[91] R[100]mm/sec CNT100;
   1:  PR[91,1] = PR[90,1] + -27.350;
   1:  PR[91,2] = PR[90,2] + -18.607;
   1:  PR[91,3] = PR[90,3] + 56.432;
   1:L PR[91] R[100]mm/sec CNT100;
   1:  PR[91,1] = PR[90,1] + -23.454;
   1:  PR[91,2] = PR[90,2] + -20.706;
   1:  PR[91,3] = PR[90,3] + 56.435;
   1:L PR[91] R[100]mm/sec CNT100;
   1:  PR[91,1] = PR[90,1] + -23.007;
   1:  PR[91,2] = PR[90,2] + -20.898;
   1:  PR[91,3] = PR[90,3] + 56.450;
   1:L PR[91] R[100]mm/sec CNT100;
   1:  PR[91,1] = PR[90,1] + -18.068;
   1:  PR[91,2] = PR[90,2] + -22.324;
   1:  PR[91,3] = PR[90,3] + 56.451;
   1:L PR[91] R[100]mm/sec CNT100;
   1:  PR[91,1] = PR[90,1] + -12.439;
   1:  PR[91,2] = PR[90,2] + -22.772;
   1:  PR[91,3] = PR[90,3] + 56.468;
   1:L PR[91] R[100]mm/sec CNT100;
   1:  PR[91,1] = PR[90,1] + -8.790;
   1:  PR[91,2] = PR[90,2] + -22.314;
   1:  PR[91,3] = PR[90,3] + 56.487;
   1:L PR[91] R[100]mm/sec CNT100;
   1:  PR[91,1] = PR[90,1] + -6.856;
   1:  PR[91,2] = PR[90,2] + -22.095;
   1:  PR[91,3] = PR[90,3] + 56.499;
   1:L PR[91] R[100]mm/sec CNT100;
   1:  PR[91,1] = PR[90,1] + -3.832;
   1:  PR[91,2] = PR[90,2] + -21.115;
   1:  PR[91,3] = PR[90,3] + 56.505;
   1:L PR[91] R[100]mm/sec CNT100;
   1:  PR[91,1] = PR[90,1] + -1.668;
   1:  PR[91,2] = PR[90,2] + -20.370;
   1:  PR[91,3] = PR[90,3] + 56.516;
   1:L PR[91] R[100]mm/sec CNT100;
   1:  PR[91,1] = PR[90,1] + 2.415;
   1:  PR[91,2] = PR[90,2] + -18.023;
   1:  PR[91,3] = PR[90,3] + 56.523;
   1:L PR[91] R[100]mm/sec CNT100;
   1:  PR[91,1] = PR[90,1] + 2.938;
   1:  PR[91,2] = PR[90,2] + -17.702;
   1:  PR[91,3] = PR[90,3] + 56.539;
   1:L PR[91] R[100]mm/sec CNT100;
   1:  PR[91,1] = PR[90,1] + 4.597;
   1:  PR[91,2] = PR[90,2] + -16.163;
   1:  PR[91,3] = PR[90,3] + 56.541;
   1:L PR[91] R[100]mm/sec CNT100;
   1:  PR[91,1] = PR[90,1] + 6.487;
   1:  PR[91,2] = PR[90,2] + -18.037;
   1:  PR[91,3] = PR[90,3] + 56.548;
   1:L PR[91] R[100]mm/sec CNT100;
   1:  PR[91,1] = PR[90,1] + 7.047;
   1:  PR[91,2] = PR[90,2] + -18.530;
   1:  PR[91,3] = PR[90,3] + 56.557;
   1:L PR[91] R[100]mm/sec CNT100;
   1:  PR[91,1] = PR[90,1] + 7.855;
   1:  PR[91,2] = PR[90,2] + -19.163;
   1:  PR[91,3] = PR[90,3] + 56.560;
   1:L PR[91] R[100]mm/sec CNT100;
   1:  PR[91,1] = PR[90,1] + 10.455;
   1:  PR[91,2] = PR[90,2] + -20.771;
   1:  PR[91,3] = PR[90,3] + 56.563;
   1:L PR[91] R[100]mm/sec CNT100;
   1:  PR[91,1] = PR[90,1] + 12.709;
   1:  PR[91,2] = PR[90,2] + -21.991;
   1:  PR[91,3] = PR[90,3] + 56.573;
   1:L PR[91] R[100]mm/sec CNT100;
   1:  PR[91,1] = PR[90,1] + 15.859;
   1:  PR[91,2] = PR[90,2] + -22.977;
   1:  PR[91,3] = PR[90,3] + 56.581;
   1:L PR[91] R[100]mm/sec CNT100;
   1:  PR[91,1] = PR[90,1] + 18.047;
   1:  PR[91,2] = PR[90,2] + -23.574;
   1:  PR[91,3] = PR[90,3] + 56.592;
   1:L PR[91] R[100]mm/sec CNT100;
   1:  PR[91,1] = PR[90,1] + 21.622;
   1:  PR[91,2] = PR[90,2] + -23.771;
